# B&R Automation Studio project Y4_V3_1 (part 6)

#### Axis2StateCyclic.ld
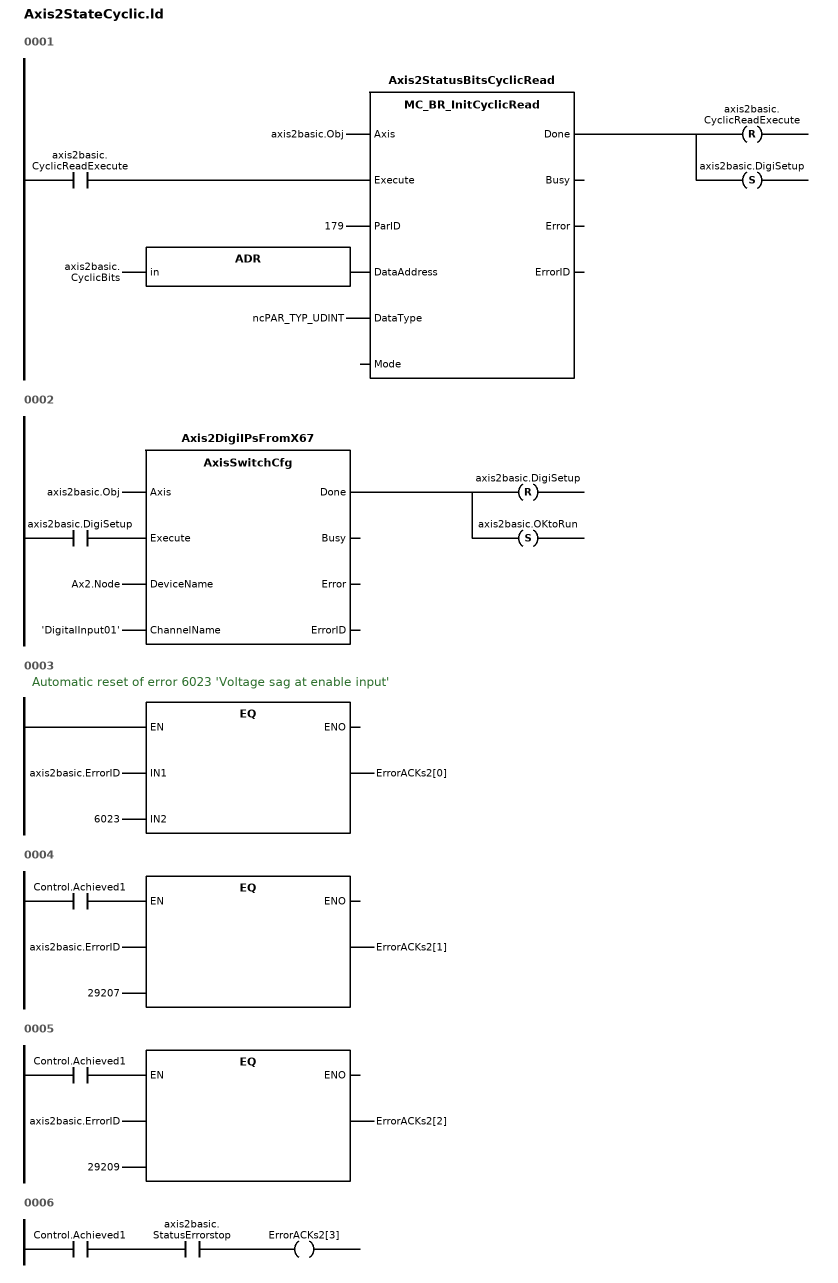
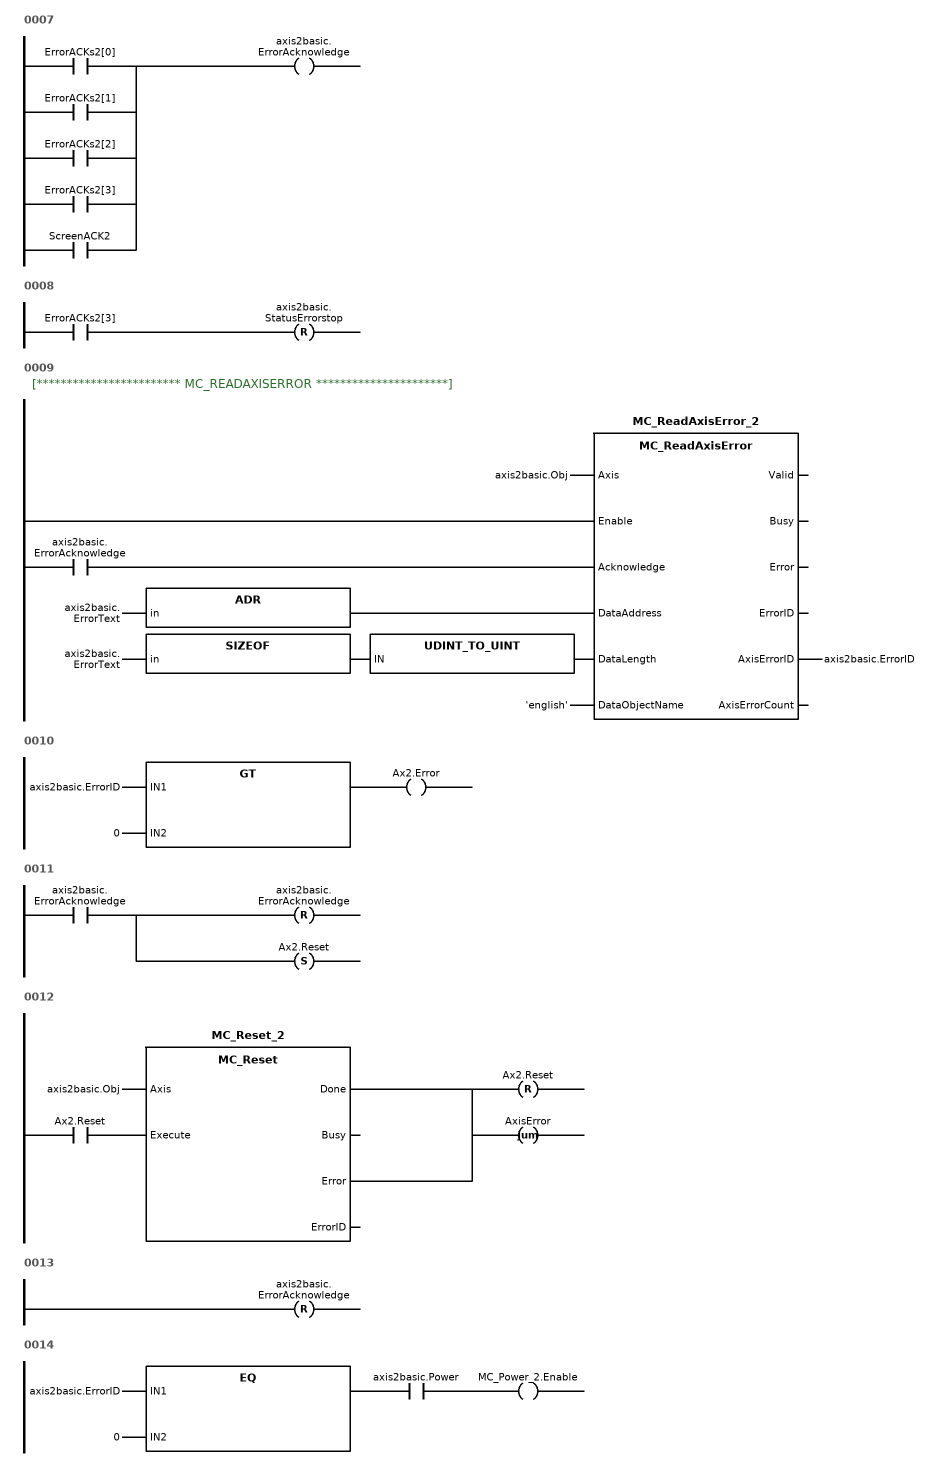
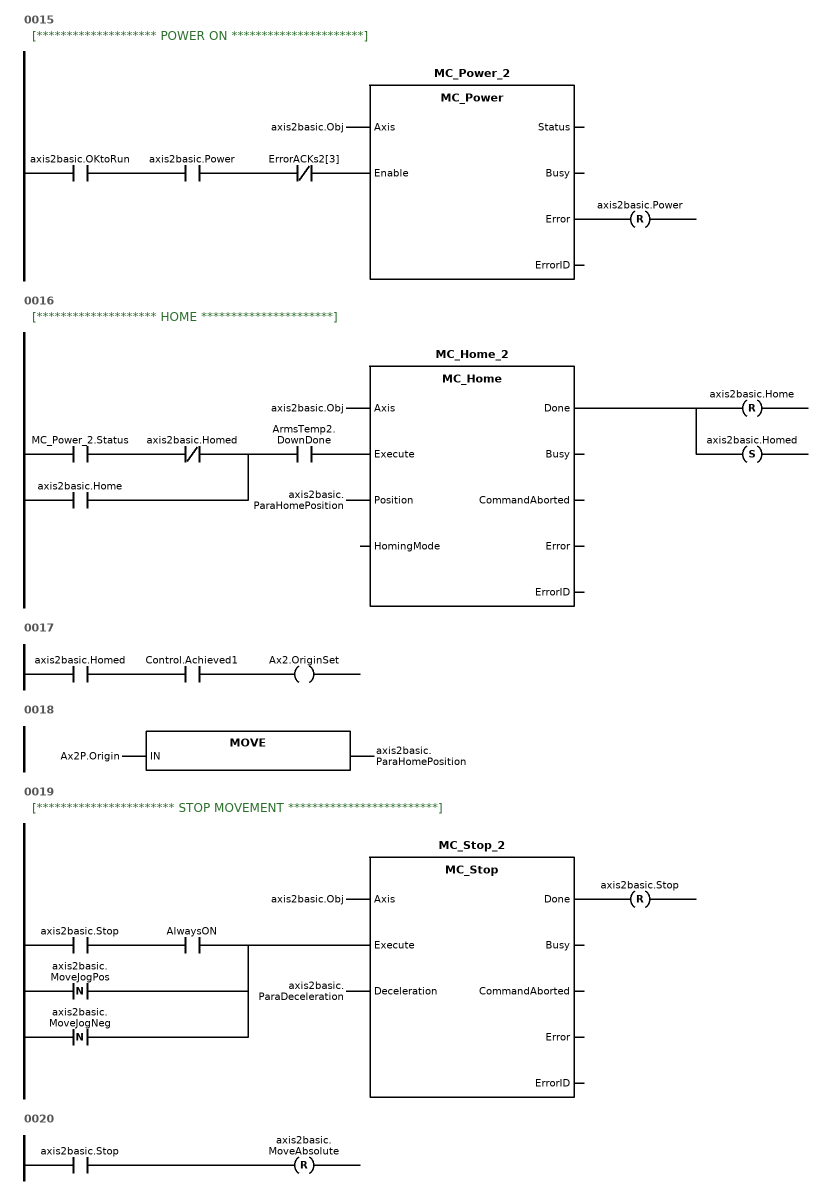
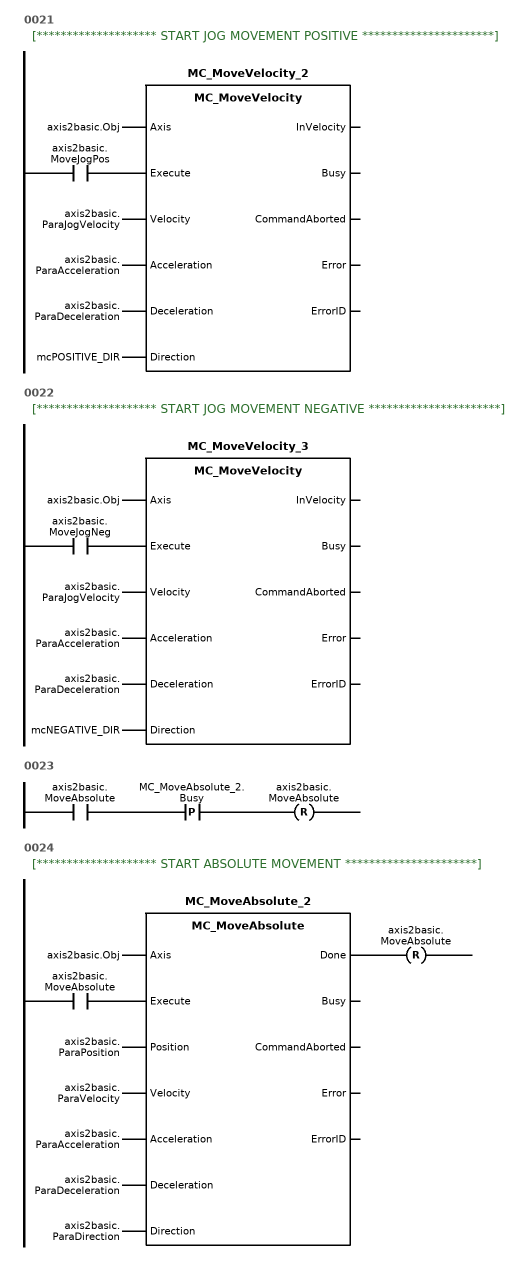
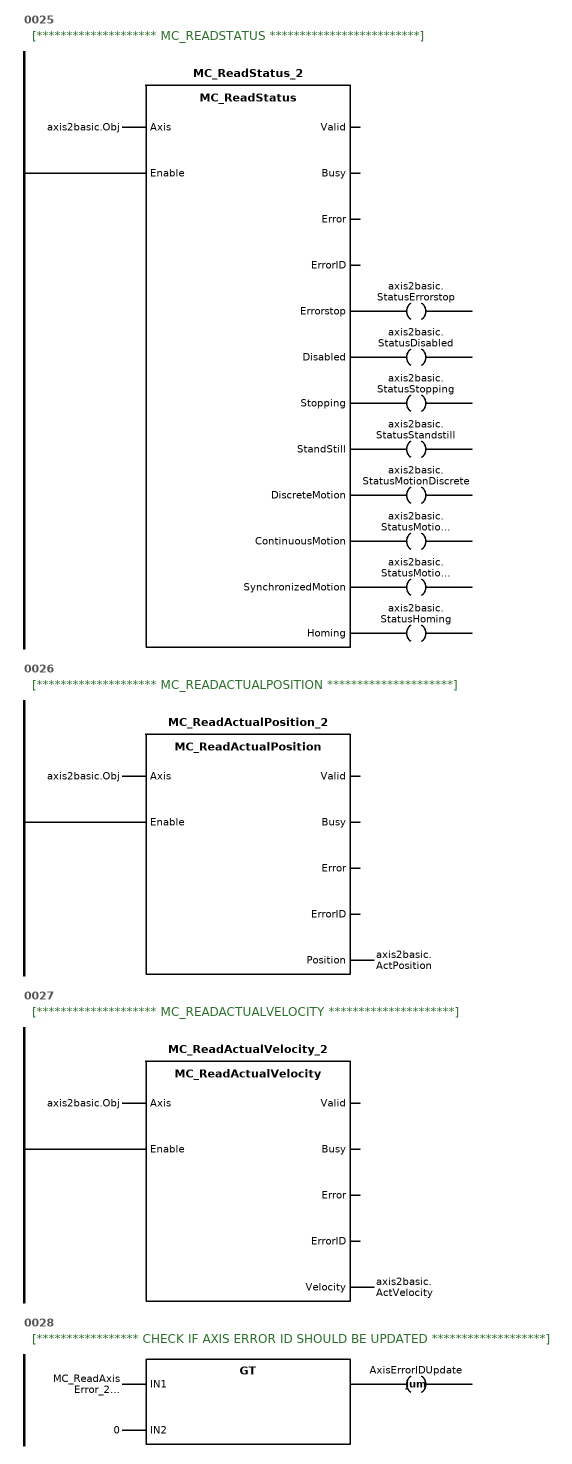
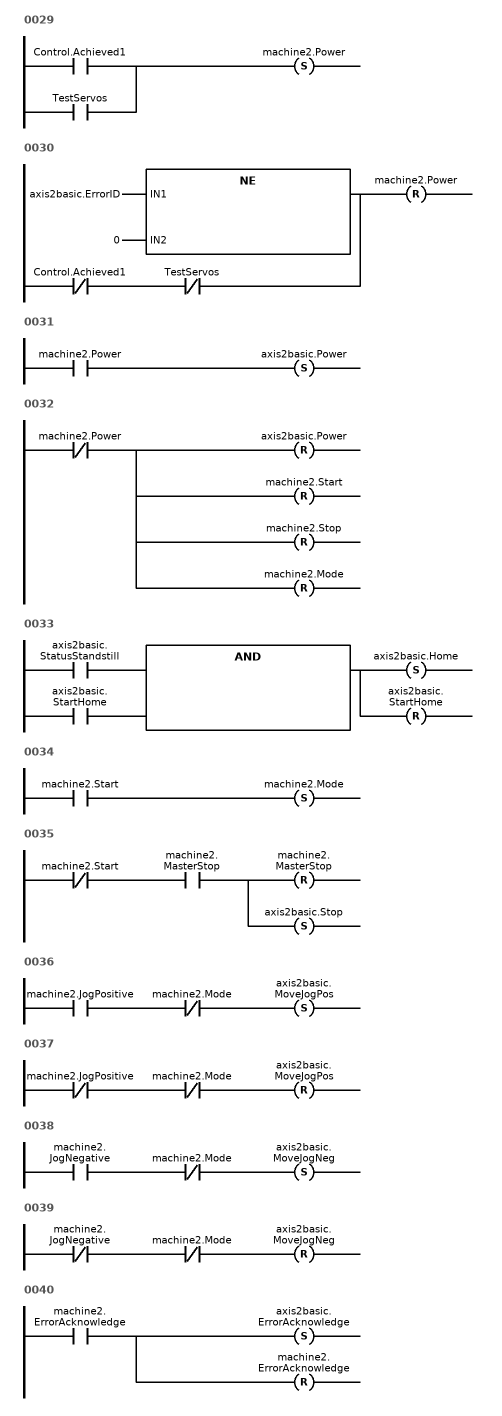
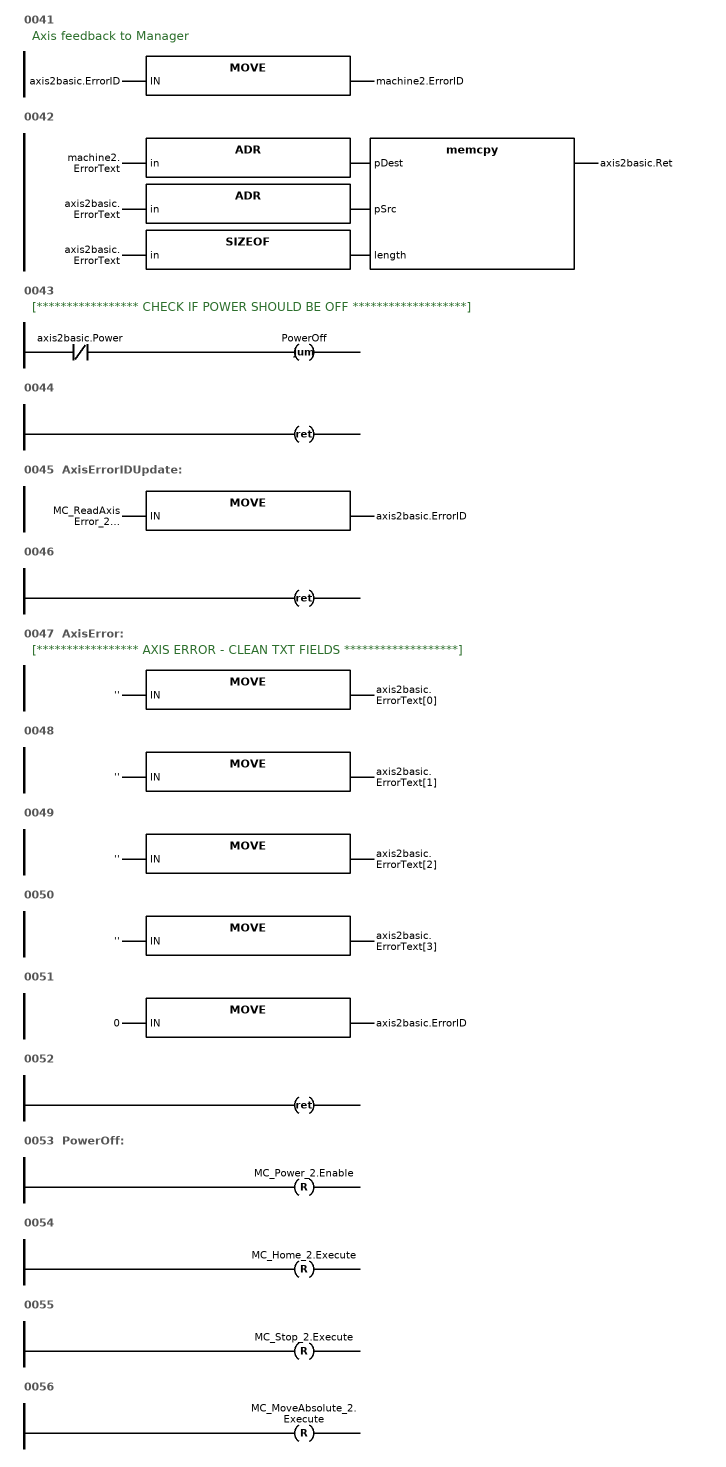
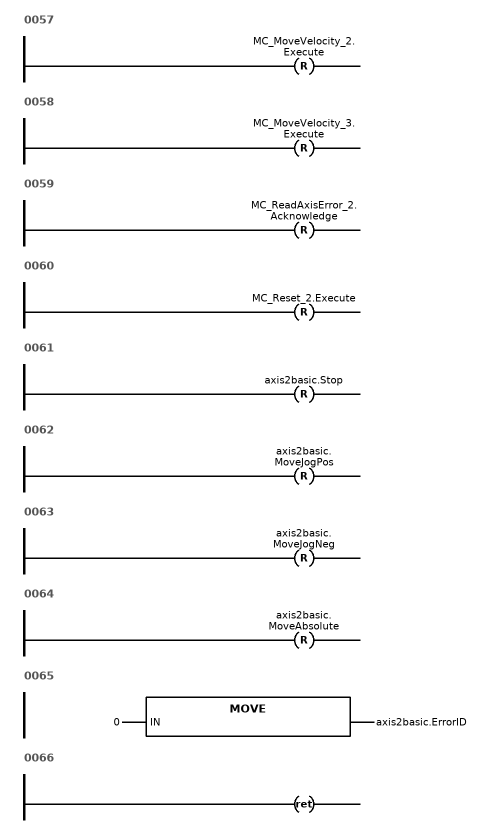
Ladder, written as Structured Text:
```iecst
PROGRAM _CYCLIC
VAR
    _p1 : BOOL;
    _e2 : F_TRIG;
    _e3 : F_TRIG;
    _e4 : R_TRIG;
    _p5 : BOOL;
    _t6 : BOOL;
    _p7 : BOOL;
END_VAR
(* Network 1 *)
Axis2StatusBitsCyclicRead(Axis := axis2basic.Obj, Execute := axis2basic.CyclicReadExecute, ParID := 179, DataAddress := ADR(in := axis2basic.CyclicBits), DataType := ncPAR_TYP_UDINT);
IF Axis2StatusBitsCyclicRead.Done THEN
    axis2basic.CyclicReadExecute := FALSE;
    axis2basic.DigiSetup := TRUE;
END_IF;

(* Network 2 *)
Axis2DigiIPsFromX67(Axis := axis2basic.Obj, Execute := axis2basic.DigiSetup, DeviceName := Ax2.Node, ChannelName := 'DigitalInput01');
IF Axis2DigiIPsFromX67.Done THEN
    axis2basic.DigiSetup := FALSE;
    axis2basic.OKtoRun := TRUE;
END_IF;

(* Network 3: Automatic reset of error 6023 'Voltage sag at enable input' *)
ErrorACKs2[0] := axis2basic.ErrorID = 6023;

(* Network 4 *)
IF Control.Achieved1 THEN ErrorACKs2[1] := axis2basic.ErrorID = 29207; END_IF;

(* Network 5 *)
IF Control.Achieved1 THEN ErrorACKs2[2] := axis2basic.ErrorID = 29209; END_IF;

(* Network 6 *)
ErrorACKs2[3] := Control.Achieved1 AND axis2basic.StatusErrorstop;

(* Network 7 *)
axis2basic.ErrorAcknowledge := ErrorACKs2[0] OR ErrorACKs2[1] OR ErrorACKs2[2] OR ErrorACKs2[3] OR ScreenACK2;

(* Network 8 *)
IF ErrorACKs2[3] THEN axis2basic.StatusErrorstop := FALSE; END_IF;

(* Network 9: [************************ MC_READAXISERROR **********************] *)
MC_ReadAxisError_2(Axis := axis2basic.Obj, Enable := TRUE, Acknowledge := axis2basic.ErrorAcknowledge, DataAddress := ADR(in := axis2basic.ErrorText), DataLength := UDINT_TO_UINT(SIZEOF(in := axis2basic.ErrorText)), DataObjectName := 'english');
axis2basic.ErrorID := MC_ReadAxisError_2.AxisErrorID;

(* Network 10 *)
Ax2.Error := axis2basic.ErrorID > 0;

(* Network 11 *)
_p1 := axis2basic.ErrorAcknowledge;
IF axis2basic.ErrorAcknowledge THEN axis2basic.ErrorAcknowledge := FALSE; END_IF;
IF _p1 THEN Ax2.Reset := TRUE; END_IF;

(* Network 12 *)
MC_Reset_2(Axis := axis2basic.Obj, Execute := Ax2.Reset);
IF MC_Reset_2.Done OR MC_Reset_2.Error THEN
    Ax2.Reset := FALSE;
    JMP AxisError;
END_IF;

(* Network 13 *)
axis2basic.ErrorAcknowledge := FALSE;

(* Network 14 *)
MC_Power_2.Enable := (axis2basic.ErrorID = 0) AND axis2basic.Power;

(* Network 15: [******************** POWER ON **********************] *)
MC_Power_2(Axis := axis2basic.Obj, Enable := axis2basic.OKtoRun AND axis2basic.Power AND NOT ErrorACKs2[3]);
IF MC_Power_2.Error THEN axis2basic.Power := FALSE; END_IF;

(* Network 16: [******************** HOME **********************] *)
MC_Home_2(Axis := axis2basic.Obj, Execute := ((MC_Power_2.Status AND NOT axis2basic.Homed) OR axis2basic.Home) AND ArmsTemp2.DownDone, Position := axis2basic.ParaHomePosition);
IF MC_Home_2.Done THEN
    axis2basic.Home := FALSE;
    axis2basic.Homed := TRUE;
END_IF;

(* Network 17 *)
Ax2.OriginSet := axis2basic.Homed AND Control.Achieved1;

(* Network 18 *)
axis2basic.ParaHomePosition := Ax2P.Origin;

(* Network 19: [*********************** STOP MOVEMENT *************************] *)
_e2(CLK := axis2basic.MoveJogPos);
_e3(CLK := axis2basic.MoveJogNeg);
MC_Stop_2(Axis := axis2basic.Obj, Execute := (axis2basic.Stop AND AlwaysON) OR _e2.Q OR _e3.Q, Deceleration := axis2basic.ParaDeceleration);
IF MC_Stop_2.Done THEN axis2basic.Stop := FALSE; END_IF;

(* Network 20 *)
IF axis2basic.Stop THEN axis2basic.MoveAbsolute := FALSE; END_IF;

(* Network 21: [******************** START JOG MOVEMENT POSITIVE **********************] *)
MC_MoveVelocity_2(Axis := axis2basic.Obj, Execute := axis2basic.MoveJogPos, Velocity := axis2basic.ParaJogVelocity, Acceleration := axis2basic.ParaAcceleration, Deceleration := axis2basic.ParaDeceleration, Direction := mcPOSITIVE_DIR);

(* Network 22: [******************** START JOG MOVEMENT NEGATIVE **********************] *)
MC_MoveVelocity_3(Axis := axis2basic.Obj, Execute := axis2basic.MoveJogNeg, Velocity := axis2basic.ParaJogVelocity, Acceleration := axis2basic.ParaAcceleration, Deceleration := axis2basic.ParaDeceleration, Direction := mcNEGATIVE_DIR);

(* Network 23 *)
_e4(CLK := MC_MoveAbsolute_2.Busy);
IF axis2basic.MoveAbsolute AND _e4.Q THEN axis2basic.MoveAbsolute := FALSE; END_IF;

(* Network 24: [******************** START ABSOLUTE MOVEMENT **********************] *)
MC_MoveAbsolute_2(Axis := axis2basic.Obj, Execute := axis2basic.MoveAbsolute, Position := axis2basic.ParaPosition, Velocity := axis2basic.ParaVelocity, Acceleration := axis2basic.ParaAcceleration, Deceleration := axis2basic.ParaDeceleration, Direction := axis2basic.ParaDirection);
IF MC_MoveAbsolute_2.Done THEN axis2basic.MoveAbsolute := FALSE; END_IF;

(* Network 25: [******************** MC_READSTATUS *************************] *)
MC_ReadStatus_2(Axis := axis2basic.Obj, Enable := TRUE);
axis2basic.StatusErrorstop := MC_ReadStatus_2.Errorstop;
axis2basic.StatusDisabled := MC_ReadStatus_2.Disabled;
axis2basic.StatusStopping := MC_ReadStatus_2.Stopping;
axis2basic.StatusStandstill := MC_ReadStatus_2.StandStill;
axis2basic.StatusMotionDiscrete := MC_ReadStatus_2.DiscreteMotion;
axis2basic.StatusMotionContinous := MC_ReadStatus_2.ContinuousMotion;
axis2basic.StatusMotionSynchronized := MC_ReadStatus_2.SynchronizedMotion;
axis2basic.StatusHoming := MC_ReadStatus_2.Homing;

(* Network 26: [******************** MC_READACTUALPOSITION *********************] *)
MC_ReadActualPosition_2(Axis := axis2basic.Obj, Enable := TRUE);
axis2basic.ActPosition := MC_ReadActualPosition_2.Position;

(* Network 27: [******************** MC_READACTUALVELOCITY *********************] *)
MC_ReadActualVelocity_2(Axis := axis2basic.Obj, Enable := TRUE);
axis2basic.ActVelocity := MC_ReadActualVelocity_2.Velocity;

(* Network 28: [***************** CHECK IF AXIS ERROR ID SHOULD BE UPDATED *******************] *)
IF MC_ReadAxisError_2.AxisErrorID > 0 THEN JMP AxisErrorIDUpdate; END_IF;

(* Network 29 *)
IF Control.Achieved1 OR TestServos THEN machine2.Power := TRUE; END_IF;

(* Network 30 *)
IF (NOT Control.Achieved1 AND NOT TestServos) OR (axis2basic.ErrorID <> 0) THEN
    machine2.Power := FALSE;
END_IF;

(* Network 31 *)
IF machine2.Power THEN axis2basic.Power := TRUE; END_IF;

(* Network 32 *)
IF NOT machine2.Power THEN axis2basic.Power := FALSE; END_IF;
_p5 := NOT machine2.Power;
IF NOT machine2.Power THEN machine2.Start := FALSE; END_IF;
IF _p5 THEN
    machine2.Stop := FALSE;
    machine2.Mode := FALSE;
END_IF;

(* Network 33 *)
_t6 := axis2basic.StatusStandstill AND axis2basic.StartHome;
IF _t6 THEN
    axis2basic.Home := TRUE;
    axis2basic.StartHome := FALSE;
END_IF;

(* Network 34 *)
IF machine2.Start THEN machine2.Mode := TRUE; END_IF;

(* Network 35 *)
_p7 := NOT machine2.Start AND machine2.MasterStop;
IF NOT machine2.Start AND machine2.MasterStop THEN machine2.MasterStop := FALSE; END_IF;
IF _p7 THEN axis2basic.Stop := TRUE; END_IF;

(* Network 36 *)
IF machine2.JogPositive AND NOT machine2.Mode THEN axis2basic.MoveJogPos := TRUE; END_IF;

(* Network 37 *)
IF NOT machine2.JogPositive AND NOT machine2.Mode THEN axis2basic.MoveJogPos := FALSE; END_IF;

(* Network 38 *)
IF machine2.JogNegative AND NOT machine2.Mode THEN axis2basic.MoveJogNeg := TRUE; END_IF;

(* Network 39 *)
IF NOT machine2.JogNegative AND NOT machine2.Mode THEN axis2basic.MoveJogNeg := FALSE; END_IF;

(* Network 40 *)
IF machine2.ErrorAcknowledge THEN
    axis2basic.ErrorAcknowledge := TRUE;
    machine2.ErrorAcknowledge := FALSE;
END_IF;

(* Network 41: Axis feedback to Manager *)
machine2.ErrorID := axis2basic.ErrorID;

(* Network 42 *)
axis2basic.Ret := memcpy(pDest := ADR(in := machine2.ErrorText), pSrc := ADR(in := axis2basic.ErrorText), length := SIZEOF(in := axis2basic.ErrorText));

(* Network 43: [***************** CHECK IF POWER SHOULD BE OFF *******************] *)
IF NOT axis2basic.Power THEN JMP PowerOff; END_IF;

(* Network 44 *)
RETURN;

(* Network 45 *)
AxisErrorIDUpdate:
axis2basic.ErrorID := MC_ReadAxisError_2.AxisErrorID;

(* Network 46 *)
RETURN;

(* Network 47: [***************** AXIS ERROR - CLEAN TXT FIELDS *******************] *)
AxisError:
axis2basic.ErrorText[0] := '';

(* Network 48 *)
axis2basic.ErrorText[1] := '';

(* Network 49 *)
axis2basic.ErrorText[2] := '';

(* Network 50 *)
axis2basic.ErrorText[3] := '';

(* Network 51 *)
axis2basic.ErrorID := 0;

(* Network 52 *)
RETURN;

(* Network 53 *)
PowerOff:
MC_Power_2.Enable := FALSE;

(* Network 54 *)
MC_Home_2.Execute := FALSE;

(* Network 55 *)
MC_Stop_2.Execute := FALSE;

(* Network 56 *)
MC_MoveAbsolute_2.Execute := FALSE;

(* Network 57 *)
MC_MoveVelocity_2.Execute := FALSE;

(* Network 58 *)
MC_MoveVelocity_3.Execute := FALSE;

(* Network 59 *)
MC_ReadAxisError_2.Acknowledge := FALSE;

(* Network 60 *)
MC_Reset_2.Execute := FALSE;

(* Network 61 *)
axis2basic.Stop := FALSE;

(* Network 62 *)
axis2basic.MoveJogPos := FALSE;

(* Network 63 *)
axis2basic.MoveJogNeg := FALSE;

(* Network 64 *)
axis2basic.MoveAbsolute := FALSE;

(* Network 65 *)
axis2basic.ErrorID := 0;

(* Network 66 *)
RETURN;
END_PROGRAM
```

### Program Logical/Motion/Axis3State (IEC)

#### Axis3StateInit.ld
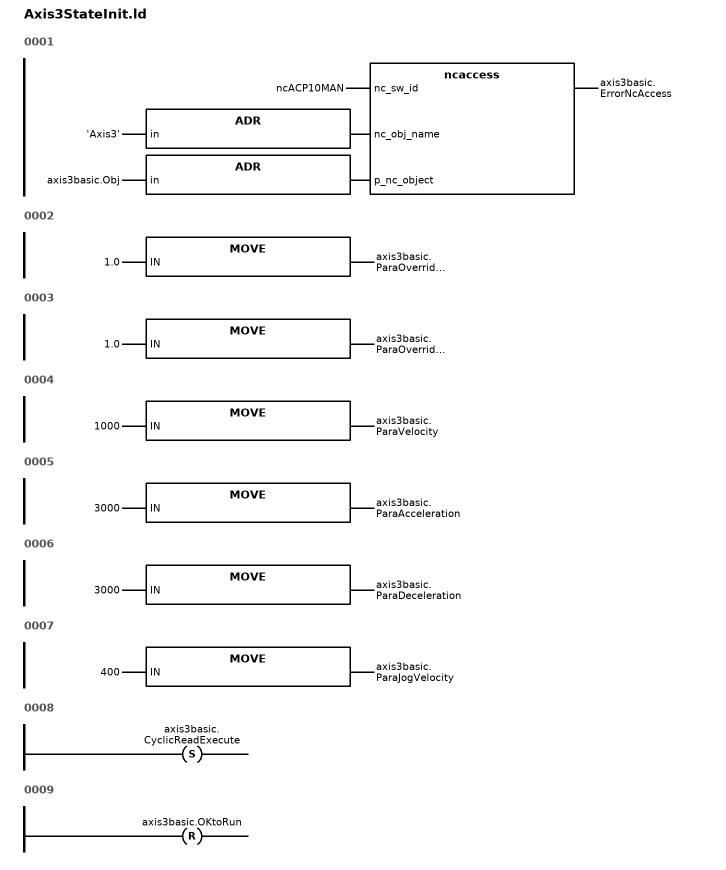
Ladder, written as Structured Text:
```iecst
PROGRAM _INIT
(* Network 1 *)
axis3basic.ErrorNcAccess := ncaccess(nc_sw_id := ncACP10MAN, nc_obj_name := ADR(in := 'Axis3'), p_nc_object := ADR(in := axis3basic.Obj));

(* Network 2 *)
axis3basic.ParaOverrideVelocity := 1.0;

(* Network 3 *)
axis3basic.ParaOverrideAcceleration := 1.0;

(* Network 4 *)
axis3basic.ParaVelocity := 1000;

(* Network 5 *)
axis3basic.ParaAcceleration := 3000;

(* Network 6 *)
axis3basic.ParaDeceleration := 3000;

(* Network 7 *)
axis3basic.ParaJogVelocity := 400;

(* Network 8 *)
axis3basic.CyclicReadExecute := TRUE;

(* Network 9 *)
axis3basic.OKtoRun := FALSE;
END_PROGRAM
```

#### Axis3StateCyclic.ld
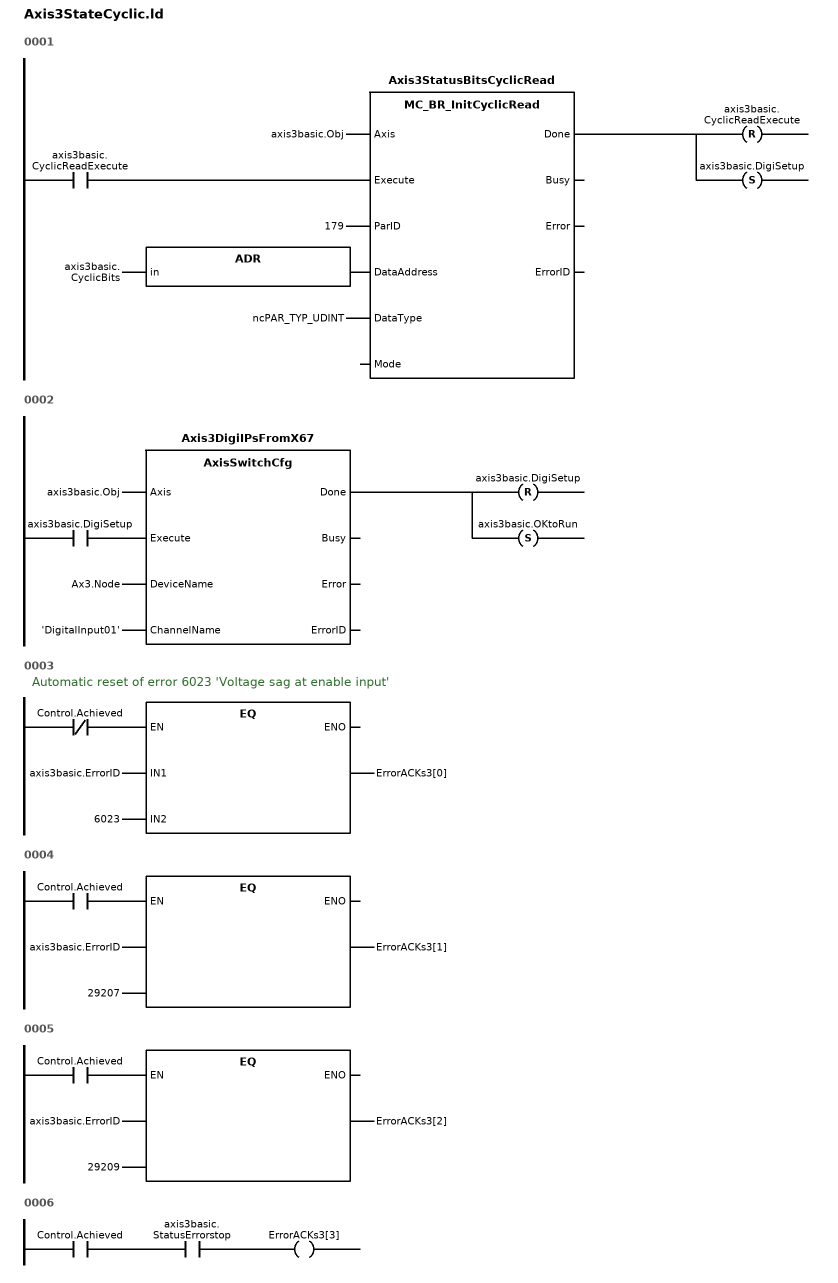
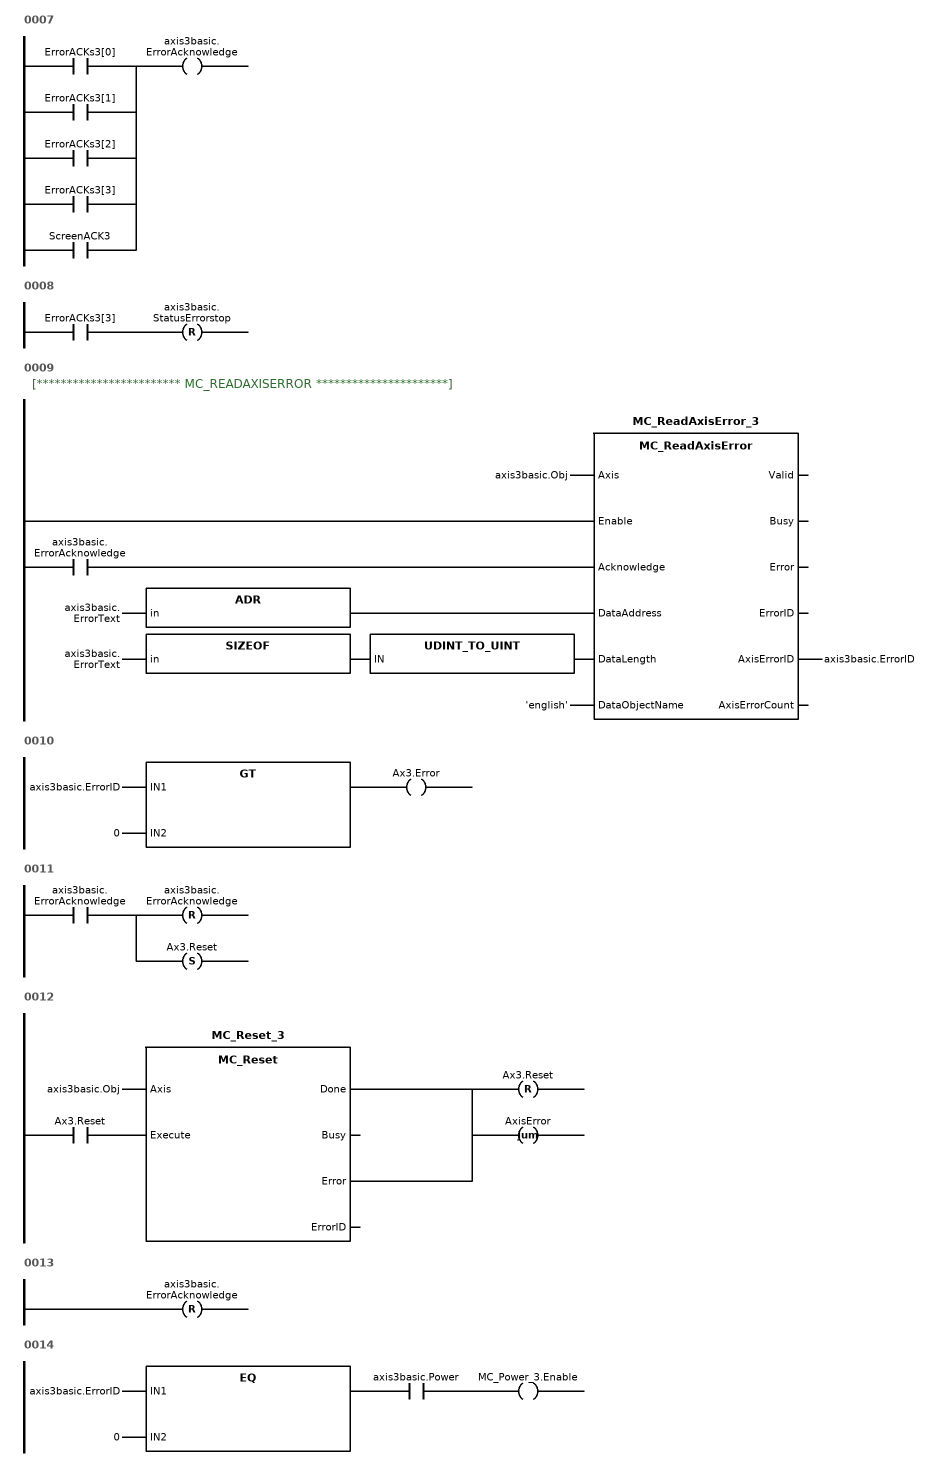
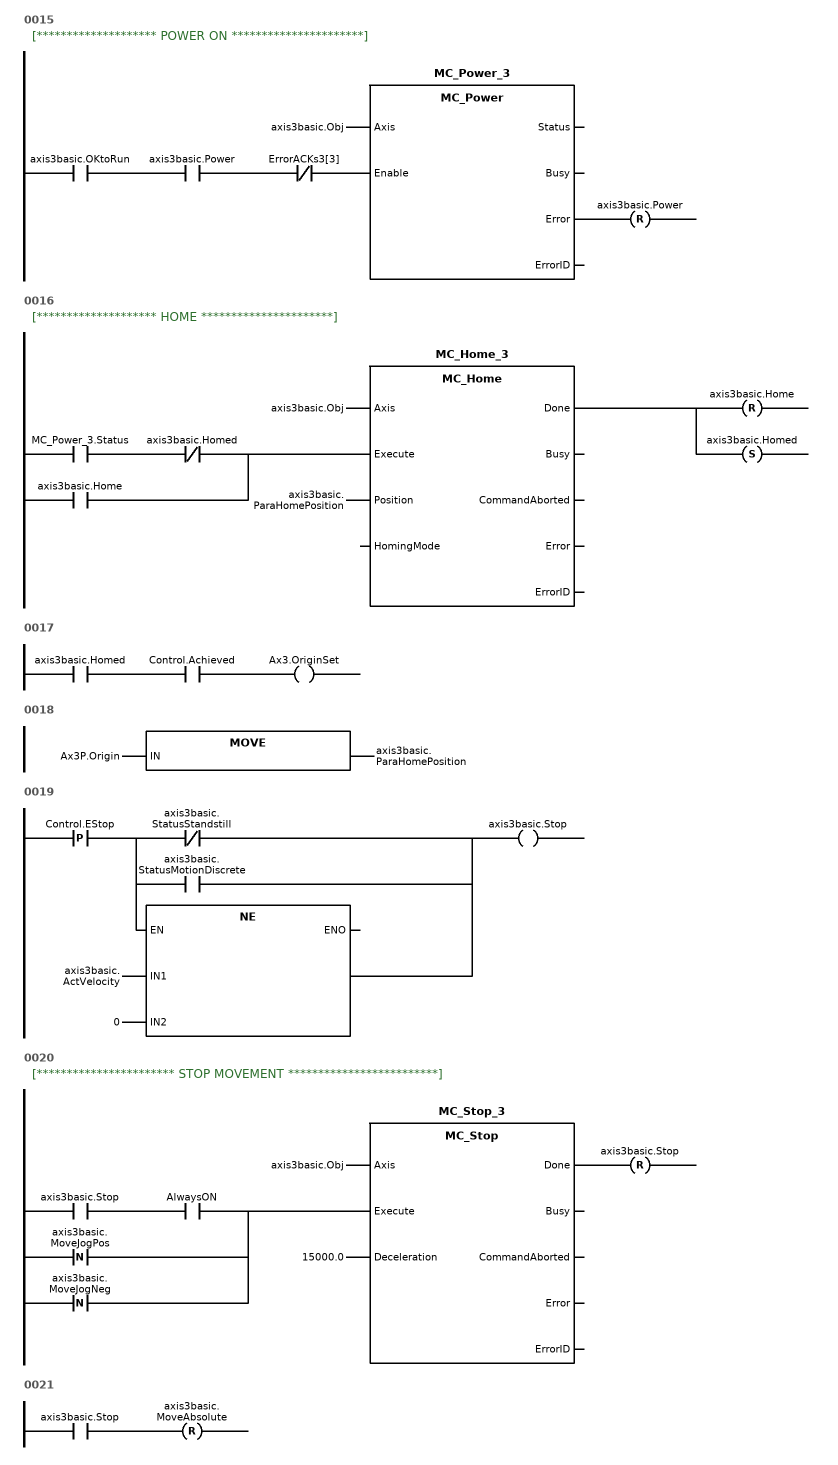
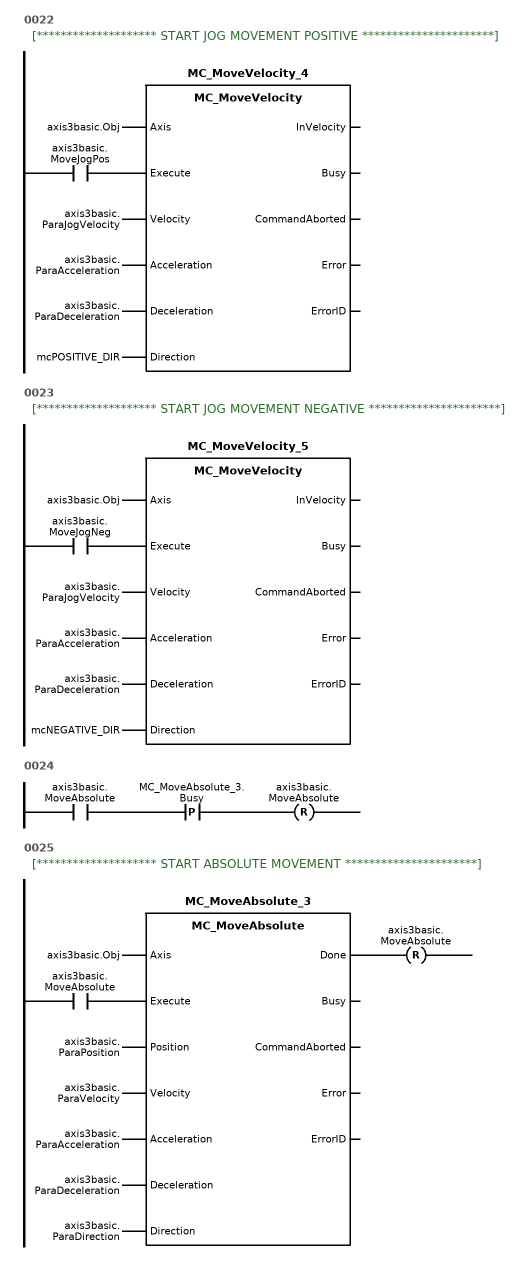
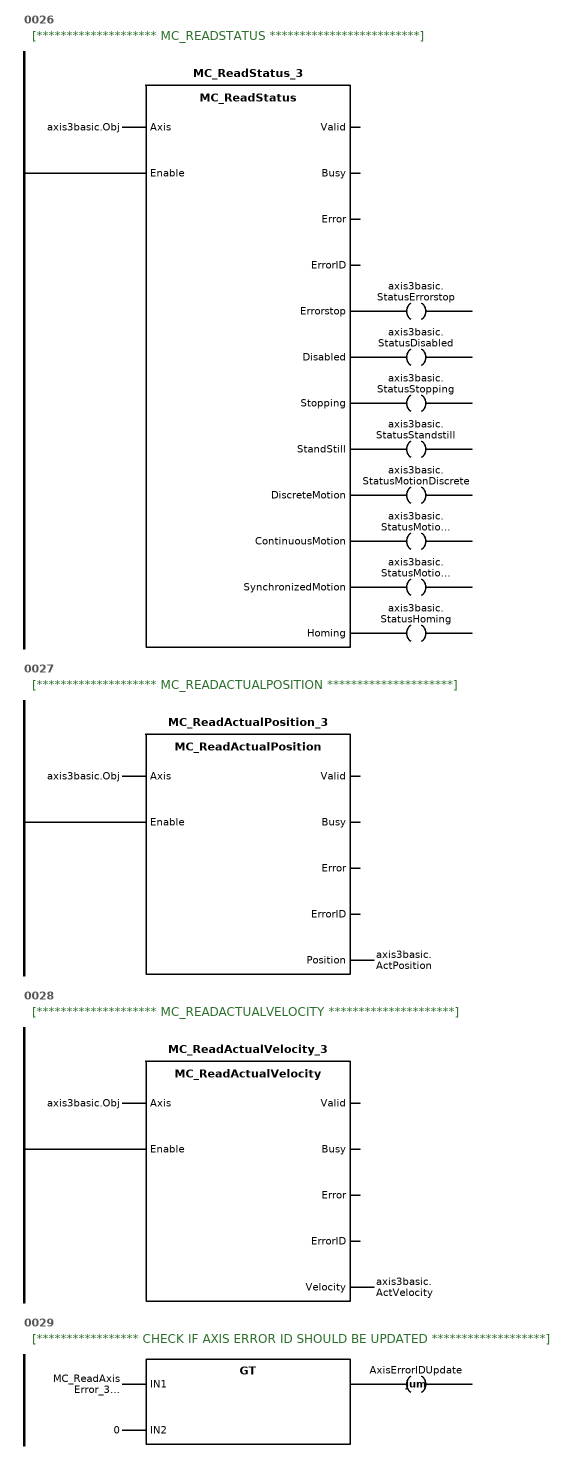
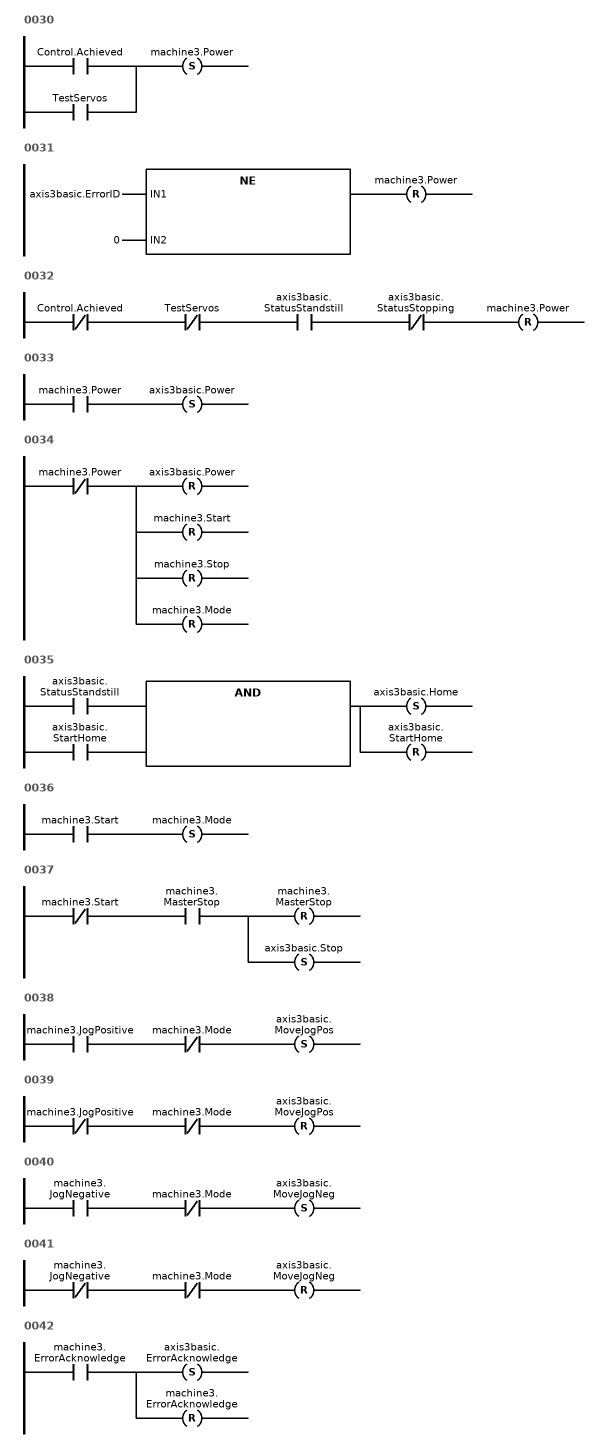
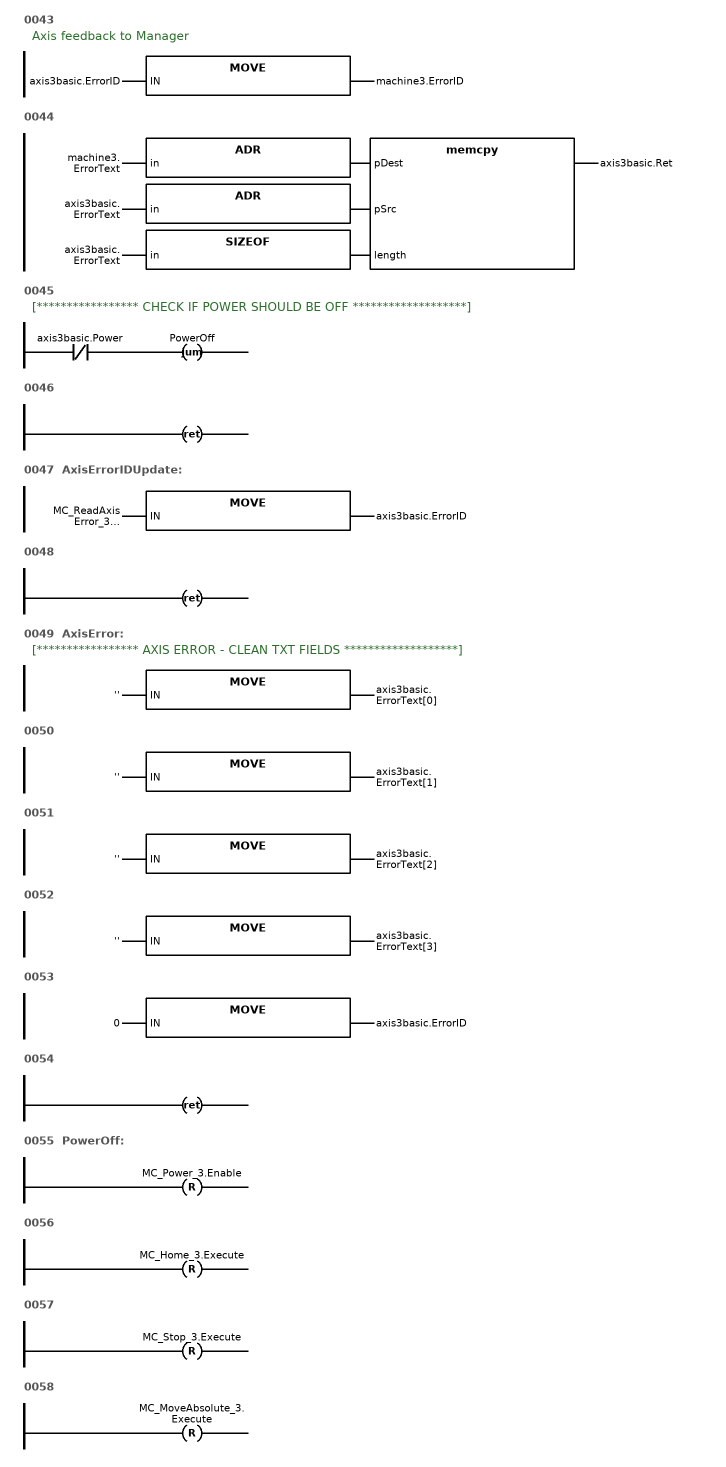
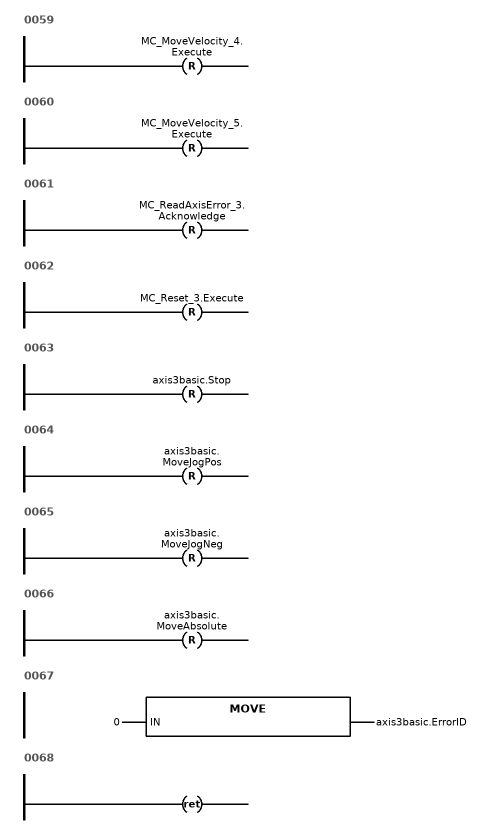
Ladder, written as Structured Text:
```iecst
PROGRAM _CYCLIC
VAR
    _p1 : BOOL;
    _e2 : R_TRIG;
    _t3 : BOOL;
    _e4 : F_TRIG;
    _e5 : F_TRIG;
    _e6 : R_TRIG;
    _p7 : BOOL;
    _t8 : BOOL;
    _p9 : BOOL;
END_VAR
(* Network 1 *)
Axis3StatusBitsCyclicRead(Axis := axis3basic.Obj, Execute := axis3basic.CyclicReadExecute, ParID := 179, DataAddress := ADR(in := axis3basic.CyclicBits), DataType := ncPAR_TYP_UDINT);
IF Axis3StatusBitsCyclicRead.Done THEN
    axis3basic.CyclicReadExecute := FALSE;
    axis3basic.DigiSetup := TRUE;
END_IF;

(* Network 2 *)
Axis3DigiIPsFromX67(Axis := axis3basic.Obj, Execute := axis3basic.DigiSetup, DeviceName := Ax3.Node, ChannelName := 'DigitalInput01');
IF Axis3DigiIPsFromX67.Done THEN
    axis3basic.DigiSetup := FALSE;
    axis3basic.OKtoRun := TRUE;
END_IF;

(* Network 3: Automatic reset of error 6023 'Voltage sag at enable input' *)
IF NOT Control.Achieved THEN ErrorACKs3[0] := axis3basic.ErrorID = 6023; END_IF;

(* Network 4 *)
IF Control.Achieved THEN ErrorACKs3[1] := axis3basic.ErrorID = 29207; END_IF;

(* Network 5 *)
IF Control.Achieved THEN ErrorACKs3[2] := axis3basic.ErrorID = 29209; END_IF;

(* Network 6 *)
ErrorACKs3[3] := Control.Achieved AND axis3basic.StatusErrorstop;

(* Network 7 *)
axis3basic.ErrorAcknowledge := ErrorACKs3[0] OR ErrorACKs3[1] OR ErrorACKs3[2] OR ErrorACKs3[3] OR ScreenACK3;

(* Network 8 *)
IF ErrorACKs3[3] THEN axis3basic.StatusErrorstop := FALSE; END_IF;

(* Network 9: [************************ MC_READAXISERROR **********************] *)
MC_ReadAxisError_3(Axis := axis3basic.Obj, Enable := TRUE, Acknowledge := axis3basic.ErrorAcknowledge, DataAddress := ADR(in := axis3basic.ErrorText), DataLength := UDINT_TO_UINT(SIZEOF(in := axis3basic.ErrorText)), DataObjectName := 'english');
axis3basic.ErrorID := MC_ReadAxisError_3.AxisErrorID;

(* Network 10 *)
Ax3.Error := axis3basic.ErrorID > 0;

(* Network 11 *)
_p1 := axis3basic.ErrorAcknowledge;
IF axis3basic.ErrorAcknowledge THEN axis3basic.ErrorAcknowledge := FALSE; END_IF;
IF _p1 THEN Ax3.Reset := TRUE; END_IF;

(* Network 12 *)
MC_Reset_3(Axis := axis3basic.Obj, Execute := Ax3.Reset);
IF MC_Reset_3.Done OR MC_Reset_3.Error THEN
    Ax3.Reset := FALSE;
    JMP AxisError;
END_IF;

(* Network 13 *)
axis3basic.ErrorAcknowledge := FALSE;

(* Network 14 *)
MC_Power_3.Enable := (axis3basic.ErrorID = 0) AND axis3basic.Power;

(* Network 15: [******************** POWER ON **********************] *)
MC_Power_3(Axis := axis3basic.Obj, Enable := axis3basic.OKtoRun AND axis3basic.Power AND NOT ErrorACKs3[3]);
IF MC_Power_3.Error THEN axis3basic.Power := FALSE; END_IF;

(* Network 16: [******************** HOME **********************] *)
MC_Home_3(Axis := axis3basic.Obj, Execute := (MC_Power_3.Status AND NOT axis3basic.Homed) OR axis3basic.Home, Position := axis3basic.ParaHomePosition);
IF MC_Home_3.Done THEN
    axis3basic.Home := FALSE;
    axis3basic.Homed := TRUE;
END_IF;

(* Network 17 *)
Ax3.OriginSet := axis3basic.Homed AND Control.Achieved;

(* Network 18 *)
axis3basic.ParaHomePosition := Ax3P.Origin;

(* Network 19 *)
_e2(CLK := Control.EStop);
IF _e2.Q THEN _t3 := axis3basic.ActVelocity <> 0; END_IF;
axis3basic.Stop := (_e2.Q AND (NOT axis3basic.StatusStandstill OR axis3basic.StatusMotionDiscrete)) OR _t3;

(* Network 20: [*********************** STOP MOVEMENT *************************] *)
_e4(CLK := axis3basic.MoveJogPos);
_e5(CLK := axis3basic.MoveJogNeg);
MC_Stop_3(Axis := axis3basic.Obj, Execute := (axis3basic.Stop AND AlwaysON) OR _e4.Q OR _e5.Q, Deceleration := 15000.0);
IF MC_Stop_3.Done THEN axis3basic.Stop := FALSE; END_IF;

(* Network 21 *)
IF axis3basic.Stop THEN axis3basic.MoveAbsolute := FALSE; END_IF;

(* Network 22: [******************** START JOG MOVEMENT POSITIVE **********************] *)
MC_MoveVelocity_4(Axis := axis3basic.Obj, Execute := axis3basic.MoveJogPos, Velocity := axis3basic.ParaJogVelocity, Acceleration := axis3basic.ParaAcceleration, Deceleration := axis3basic.ParaDeceleration, Direction := mcPOSITIVE_DIR);

(* Network 23: [******************** START JOG MOVEMENT NEGATIVE **********************] *)
MC_MoveVelocity_5(Axis := axis3basic.Obj, Execute := axis3basic.MoveJogNeg, Velocity := axis3basic.ParaJogVelocity, Acceleration := axis3basic.ParaAcceleration, Deceleration := axis3basic.ParaDeceleration, Direction := mcNEGATIVE_DIR);

(* Network 24 *)
_e6(CLK := MC_MoveAbsolute_3.Busy);
IF axis3basic.MoveAbsolute AND _e6.Q THEN axis3basic.MoveAbsolute := FALSE; END_IF;

(* Network 25: [******************** START ABSOLUTE MOVEMENT **********************] *)
MC_MoveAbsolute_3(Axis := axis3basic.Obj, Execute := axis3basic.MoveAbsolute, Position := axis3basic.ParaPosition, Velocity := axis3basic.ParaVelocity, Acceleration := axis3basic.ParaAcceleration, Deceleration := axis3basic.ParaDeceleration, Direction := axis3basic.ParaDirection);
IF MC_MoveAbsolute_3.Done THEN axis3basic.MoveAbsolute := FALSE; END_IF;

(* Network 26: [******************** MC_READSTATUS *************************] *)
MC_ReadStatus_3(Axis := axis3basic.Obj, Enable := TRUE);
axis3basic.StatusErrorstop := MC_ReadStatus_3.Errorstop;
axis3basic.StatusDisabled := MC_ReadStatus_3.Disabled;
axis3basic.StatusStopping := MC_ReadStatus_3.Stopping;
axis3basic.StatusStandstill := MC_ReadStatus_3.StandStill;
axis3basic.StatusMotionDiscrete := MC_ReadStatus_3.DiscreteMotion;
axis3basic.StatusMotionContinous := MC_ReadStatus_3.ContinuousMotion;
axis3basic.StatusMotionSynchronized := MC_ReadStatus_3.SynchronizedMotion;
axis3basic.StatusHoming := MC_ReadStatus_3.Homing;

(* Network 27: [******************** MC_READACTUALPOSITION *********************] *)
MC_ReadActualPosition_3(Axis := axis3basic.Obj, Enable := TRUE);
axis3basic.ActPosition := MC_ReadActualPosition_3.Position;

(* Network 28: [******************** MC_READACTUALVELOCITY *********************] *)
MC_ReadActualVelocity_3(Axis := axis3basic.Obj, Enable := TRUE);
axis3basic.ActVelocity := MC_ReadActualVelocity_3.Velocity;

(* Network 29: [***************** CHECK IF AXIS ERROR ID SHOULD BE UPDATED *******************] *)
IF MC_ReadAxisError_3.AxisErrorID > 0 THEN JMP AxisErrorIDUpdate; END_IF;

(* Network 30 *)
IF Control.Achieved OR TestServos THEN machine3.Power := TRUE; END_IF;

(* Network 31 *)
IF axis3basic.ErrorID <> 0 THEN machine3.Power := FALSE; END_IF;

(* Network 32 *)
IF NOT Control.Achieved AND NOT TestServos AND axis3basic.StatusStandstill AND NOT axis3basic.StatusStopping THEN
    machine3.Power := FALSE;
END_IF;

(* Network 33 *)
IF machine3.Power THEN axis3basic.Power := TRUE; END_IF;

(* Network 34 *)
IF NOT machine3.Power THEN axis3basic.Power := FALSE; END_IF;
_p7 := NOT machine3.Power;
IF NOT machine3.Power THEN machine3.Start := FALSE; END_IF;
IF _p7 THEN
    machine3.Stop := FALSE;
    machine3.Mode := FALSE;
END_IF;

(* Network 35 *)
_t8 := axis3basic.StatusStandstill AND axis3basic.StartHome;
IF _t8 THEN
    axis3basic.Home := TRUE;
    axis3basic.StartHome := FALSE;
END_IF;

(* Network 36 *)
IF machine3.Start THEN machine3.Mode := TRUE; END_IF;

(* Network 37 *)
_p9 := NOT machine3.Start AND machine3.MasterStop;
IF NOT machine3.Start AND machine3.MasterStop THEN machine3.MasterStop := FALSE; END_IF;
IF _p9 THEN axis3basic.Stop := TRUE; END_IF;

(* Network 38 *)
IF machine3.JogPositive AND NOT machine3.Mode THEN axis3basic.MoveJogPos := TRUE; END_IF;

(* Network 39 *)
IF NOT machine3.JogPositive AND NOT machine3.Mode THEN axis3basic.MoveJogPos := FALSE; END_IF;

(* Network 40 *)
IF machine3.JogNegative AND NOT machine3.Mode THEN axis3basic.MoveJogNeg := TRUE; END_IF;

(* Network 41 *)
IF NOT machine3.JogNegative AND NOT machine3.Mode THEN axis3basic.MoveJogNeg := FALSE; END_IF;

(* Network 42 *)
IF machine3.ErrorAcknowledge THEN
    axis3basic.ErrorAcknowledge := TRUE;
    machine3.ErrorAcknowledge := FALSE;
END_IF;

(* Network 43: Axis feedback to Manager *)
machine3.ErrorID := axis3basic.ErrorID;

(* Network 44 *)
axis3basic.Ret := memcpy(pDest := ADR(in := machine3.ErrorText), pSrc := ADR(in := axis3basic.ErrorText), length := SIZEOF(in := axis3basic.ErrorText));

(* Network 45: [***************** CHECK IF POWER SHOULD BE OFF *******************] *)
IF NOT axis3basic.Power THEN JMP PowerOff; END_IF;

(* Network 46 *)
RETURN;

(* Network 47 *)
AxisErrorIDUpdate:
axis3basic.ErrorID := MC_ReadAxisError_3.AxisErrorID;

(* Network 48 *)
RETURN;

(* Network 49: [***************** AXIS ERROR - CLEAN TXT FIELDS *******************] *)
AxisError:
axis3basic.ErrorText[0] := '';

(* Network 50 *)
axis3basic.ErrorText[1] := '';

(* Network 51 *)
axis3basic.ErrorText[2] := '';

(* Network 52 *)
axis3basic.ErrorText[3] := '';

(* Network 53 *)
axis3basic.ErrorID := 0;

(* Network 54 *)
RETURN;

(* Network 55 *)
PowerOff:
MC_Power_3.Enable := FALSE;

(* Network 56 *)
MC_Home_3.Execute := FALSE;

(* Network 57 *)
MC_Stop_3.Execute := FALSE;

(* Network 58 *)
MC_MoveAbsolute_3.Execute := FALSE;

(* Network 59 *)
MC_MoveVelocity_4.Execute := FALSE;

(* Network 60 *)
MC_MoveVelocity_5.Execute := FALSE;

(* Network 61 *)
MC_ReadAxisError_3.Acknowledge := FALSE;

(* Network 62 *)
MC_Reset_3.Execute := FALSE;

(* Network 63 *)
axis3basic.Stop := FALSE;

(* Network 64 *)
axis3basic.MoveJogPos := FALSE;

(* Network 65 *)
axis3basic.MoveJogNeg := FALSE;

(* Network 66 *)
axis3basic.MoveAbsolute := FALSE;

(* Network 67 *)
axis3basic.ErrorID := 0;

(* Network 68 *)
RETURN;
END_PROGRAM
```

### Data object Logical/Motion/axis3 (Ax) - ACP10: Axis data object.

#### axis3.ax
```
InitParameter (Version=2.37.0, NcSwId=ACP10)
  ACP10AXIS_typ:
    dig_in:
      level:
        reference = ncACTIV_HI
        pos_hw_end = ncACTIV_LO
        neg_hw_end = ncACTIV_LO
        trigger1 = ncACTIV_HI
        trigger2 = ncACTIV_HI
    encoder_if:
      parameter:
        count_dir = ncSTANDARD
        scaling:
          load:
            units = 1521
            rev_motor = 10
    limit:
      parameter:
        v_pos = 10000
        v_neg = 10000
        a1_pos = 9000.0
        a2_pos = 7000.0
        a1_neg = 9000.0
        a2_neg = 7000.0
        t_jolt = 0
        t_in_pos = 0
        pos_sw_end = 2000000000
        neg_sw_end = -2000000000
        ds_warning = 500
        ds_stop = 1000
        a_stop = 1.0e30
        dv_stop = 0
        dv_stop_mode = ncOFF
    controller:
      mode = ncPOSITION
      position:
        kv = 50
        tn = 0
        t_predict = 0.0008
        t_total = 0.0008
        p_max = 10000
        i_max = 0
      speed:
        kv = 2.0
        tn = 0
        t_filter = 0.0
        isq_filter1:
          type = ncOFF
          a0 = 0.0
          a1 = 0.0
          b0 = 0.0
          b1 = 0.0
          b2 = 0.0
          c0_par_id = 0
          c1_par_id = 0
        isq_filter2:
          type = ncOFF
          a0 = 0.0
          a1 = 0.0
          b0 = 0.0
          b1 = 0.0
          b2 = 0.0
          c0_par_id = 0
          c1_par_id = 0
        isq_filter3:
          type = ncOFF
          a0 = 0.0
          a1 = 0.0
          b0 = 0.0
          b1 = 0.0
          b2 = 0.0
          c0_par_id = 0
          c1_par_id = 0
      uf:
        type = ncLINEAR
        auto_config = ncMOTOR_PAR
        u0 = 0
        un = 0
        fn = 50.0
        k_f_slip = 0
      ff:
        torque_load = 0.0
        torque_pos = 0.0
        torque_neg = 0.0
        kv_torque = 0.0
        inertia = 0.0
        t_filter_a = 0.0
    move:
      stop:
        parameter[0]:
          decel_ramp = ncA_LIMIT
          controller = ncON
        parameter[1]:
          decel_ramp = ncA_LIMIT
          controller = ncON
        parameter[2]:
          decel_ramp = ncA_LIMIT
          controller = ncON
        parameter[3]:
          decel_ramp = ncA_LIMIT
          controller = ncON
        quickstop:
          decel_ramp = ncA_LIMIT
        drive_error:
          decel_ramp = ncA_LIMIT
      homing:
        parameter:
          s = 0
          v_switch = 500.0
          v_trigger = 25.0
          a = 1000.0
          mode = ncSWITCH_GATE
          edge_sw = ncNEGATIVE
          start_dir = ncNEGATIVE
          trigg_dir = ncNEGATIVE
          ref_pulse = ncOFF
          fix_dir = ncOFF
          tr_s_block = 0
          torque_lim = 0
          ds_block = 0
          ds_stop = 0
      basis:
        parameter:
          v_pos = 10000
          v_neg = 10000
          a1_pos = 50000
          a2_pos = 40000.0
          a1_neg = 50000
          a2_neg = 40000.0
    message:
      text:
        parameter:
          format = ncBREAK
          columns = 80
          data_modul = english
```

### Data object Logical/Motion/table_par3 (Apt) - ACOPOS Parameter Table

#### table_par3.apt
```
AcoposParameterTable:
  Root Parameters:
    8JSA54.R0050D000-0 Rev.C0 (StructureEdit=FALSE)  // 8JSA54.R0050D000-0 Rev.C0
      General parameters:
        30 = 0x0002 (Name=MOTOR_TYPE)  // Motor: Type
        31 = 0x0203 (Name=MOTOR_COMPATIBILITY)  // Motor: Software compatibility
        46 = 1 (Name=MOTOR_WIND_CONNECT)  // Motor: Winding connection
        47 = 5 (Name=MOTOR_POLEPAIRS)  // Motor: Number of pole-pairs
      Brake parameters:
        42 = 0 (Name=MOTOR_BRAKE_CURR_RATED, Unit=A)  // Motor holding brake: Rated current
        43 = 0 (Name=MOTOR_BRAKE_TORQ_RATED, Unit=Nm)  // Motor holding brake: Rated torque
        44 = 0 (Name=MOTOR_BRAKE_ON_TIME, Unit=s)  // Motor holding brake: Engaging delay
        45 = 0 (Name=MOTOR_BRAKE_OFF_TIME, Unit=s)  // Motor holding brake: Release delay
      Thermo sensor parameters:
        64 = 632 (Name=MOTOR_TEMPSENS_PAR1)  // Temperature sensor: Parameter 1
        65 = 2225 (Name=MOTOR_TEMPSENS_PAR2)  // Temperature sensor: Parameter 2
        66 = -30 (Name=MOTOR_TEMPSENS_PAR3)  // Temperature sensor: Parameter 3
        67 = 5.7266 (Name=MOTOR_TEMPSENS_PAR4)  // Temperature sensor: Parameter 4
        68 = 36.0938 (Name=MOTOR_TEMPSENS_PAR5)  // Temperature sensor: Parameter 5
        69 = 62.9375 (Name=MOTOR_TEMPSENS_PAR6)  // Temperature sensor: Parameter 6
        70 = 87.25 (Name=MOTOR_TEMPSENS_PAR7)  // Temperature sensor: Parameter 7
        71 = 109.6016 (Name=MOTOR_TEMPSENS_PAR8)  // Temperature sensor: Parameter 8
        72 = 130.3984 (Name=MOTOR_TEMPSENS_PAR9)  // Temperature sensor: Parameter 9
        73 = 150 (Name=MOTOR_TEMPSENS_PAR10)  // Temperature sensor: Parameter 10
        75 = 0 (Name=MOTOR_THERMAL_CONST, Unit=s)  // Motor: Thermal time constant (for MOTOR_COMPATIBILITY 0x0202)
      Motor parameters:
        48 = 560 (Name=MOTOR_VOLTAGE_RATED, Unit=V)  // Motor: Rated voltage
        49 = 73.3 (Name=MOTOR_VOLTAGE_CONST, Unit=mV*min)  // Motor: Voltage constant
        50 = 5000 (Name=MOTOR_SPEED_RATED, Unit=1/min)  // Motor: Rated speed
        51 = 6000 (Name=MOTOR_SPEED_MAX, Unit=1/min)  // Motor: Maximum speed
        52 = 14.1 (Name=MOTOR_TORQ_STALL, Unit=Nm)  // Motor: Stall torque
        53 = 6.92 (Name=MOTOR_TORQ_RATED, Unit=Nm)  // Motor: Rated torque
        54 = 53.7 (Name=MOTOR_TORQ_MAX, Unit=Nm)  // Motor: Peak torque
        55 = 1.13 (Name=MOTOR_TORQ_CONST, Unit=Nm/A)  // Motor: Torque constant
        56 = 12.5 (Name=MOTOR_CURR_STALL, Unit=A)  // Motor: Stall current
        57 = 6.11 (Name=MOTOR_CURR_RATED, Unit=A)  // Motor: Rated current
        58 = 62.5 (Name=MOTOR_CURR_MAX, Unit=A)  // Motor: Peak current
        59 = 1.2973 (Name=MOTOR_WIND_CROSS_SECT, Unit=mm²)  // Motor: Line cross section
        60 = 0.65 (Name=MOTOR_STATOR_RESISTANCE, Unit=Ohm)  // Motor: Stator resistance
        61 = 0.0035 (Name=MOTOR_STATOR_INDUCTANCE, Unit=Henry)  // Motor: Stator inductance
        62 = 0.0012 (Name=MOTOR_INERTIA, Unit=kgm²)  // Motor: Moment of inertia
        63 = 0 (Name=MOTOR_COMMUT_OFFSET, Unit=rad)  // Motor: Commutation offset
        849 = 1860 (Name=MOTOR_TAU_THERM, Unit=s)  // Motor: Thermal time constant
      Isolation parameters:
        74 = 130 (Name=MOTOR_WIND_TEMP_MAX, Unit=°C)  // Temperature sensor: Limit temperature
    SS2 (StructureEdit=FALSE)  // 8AC122.60-3
      97 = ncRESOLVER (Name=ENCOD_TYPE)  // Encoder1: Type
      109 = 4096 (Name=SCALE_ENCOD_INCR)  // Encoder1: Encoder scaling: increments per SCALE_ENCOD_MOTOR_REV motor revolutions
      203 = 1 (Name=ENCOD_POLEPAIRS)  // Encoder1: Resolver polepairs per encoder revolution
      727 = 0 (Name=ENCOD_LINE_CHK_IGNORE)  // Encoder1: Ignore check
      1048 = 0.5 (Name=ENCOD_TRANS_RATIO)  // Encoder1: Resolver transmission ratio
```

### IPConfig.var - Local variables
```iecst
(********************************************************************
 * COPYRIGHT --
 ********************************************************************
 * Program: IPConfig
 * File: IPConfig.var
 * Author: wallisj
 * Created: July 17, 2008
 ********************************************************************
 * Local variables of program IPConfig
 ********************************************************************)
VAR
	ActBroadcastAddr : STRING[16];
	ActDefaultGateway : STRING[16];
	ActIPAddr : STRING[16];
	ActSubnetMask : STRING[16];
	CfgGetBroadcastAddr_0 : CfgGetBroadcastAddr;
	CfgGetDefaultGateway_0 : CfgGetDefaultGateway;
	CfgGetInaNode_0 : CfgGetInaNode;
	CfgGetIPAddr_0 : CfgGetIPAddr;
	CfgGetSubnetMask_0 : CfgGetSubnetMask;
	CfgSetBroadcastAddr_0 : CfgSetBroadcastAddr;
	CfgSetDefaultGateway_0 : CfgSetDefaultGateway;
	CfgSetIPAddr_0 : CfgSetIPAddr;
	CfgSetSubnetMask_0 : CfgSetSubnetMask;
	InaNodeNumber : USINT;
	ReadBroadcastAddr : BOOL;
	ReadBroadcastAddrError : UINT;
	ReadDefaultGateway : BOOL;
	ReadDefaultGatewayError : UINT;
	ReadEthernetSettings : BOOL;
	ReadInaNode : BOOL;
	ReadInaNodeError : UINT;
	ReadIPAddr : BOOL;
	ReadIPAddrError : UINT := 0;
	ReadSubnetMask : BOOL;
	ReadSubnetMaskError : UINT;
	ReBoot : BOOL;
	SetBroadcastAddr : STRING[16];
	SetDefaultGateway : STRING[16];
	SetIPAddr : STRING[16];
	SetSubnetMask : STRING[16];
	WriteBroadcastAddr : BOOL;
	WriteBroadcastAddrError : UINT;
	WriteDefaultGateway : BOOL;
	WriteDefaultGatewayError : UINT;
	WriteEthernetSettings : BOOL;
	WriteIPAddr : BOOL;
	WriteIPAddrError : UINT;
	WriteSubnetMask : BOOL;
	WriteSubnetMaskError : UINT;
END_VAR
```

### Program Logical/IPConfig/IPConfig (IEC) - Ethernet settings read/write

#### IPConfigInit.st - Initialization code
```iecst
(********************************************************************
 * COPYRIGHT --
 ********************************************************************
 * Program: IPConfig
 * File: IPConfigInit.st
 * Author: wallisj
 * Created: July 17, 2008
 ********************************************************************
 * Implementation of program IPConfig
 ********************************************************************)

PROGRAM _INIT

	ReadEthernetSettings := TRUE;

END_PROGRAM
```

#### IPConfigCyclic.st - Cyclic code
```iecst
(********************************************************************
 * COPYRIGHT --
 ********************************************************************
 * Program: IPConfig
 * File: IPConfigCyclic.st
 * Author: wallisj
 * Created: July 17, 2008
 ********************************************************************
 * Implementation of program IPConfig
 ********************************************************************)

PROGRAM _CYCLIC

(*----------------------------------------------------------------------------------*)
(* Flag control for reading the Ethernet settings									*)
(*----------------------------------------------------------------------------------*)
	IF (ReadEthernetSettings = TRUE) THEN
 		ReadInaNode 			:= TRUE;
		ReadIPAddr				:= TRUE;
		ReadSubnetMask			:= TRUE;
		ReadDefaultGateway		:= TRUE;
		ReadBroadcastAddr		:= TRUE;
		ReadEthernetSettings	:= FALSE;
	END_IF

(*----------------------------------------------------------------------------------*)
(* Flag control for writing the Ethernet settings									*)
(*----------------------------------------------------------------------------------*)
	IF (WriteEthernetSettings = TRUE) THEN
 		WriteIPAddr				:= TRUE;
		WriteSubnetMask			:= TRUE;
		WriteDefaultGateway		:= TRUE;
		WriteBroadcastAddr		:= TRUE;
		WriteEthernetSettings	:= FALSE;
	END_IF

(*----------------------------------------------------------------------------------*)
(* Read in the INA node number														*)
(*----------------------------------------------------------------------------------*)
	CfgGetInaNode_0.enable 		:= ReadInaNode;
	CfgGetInaNode_0.pDevice 	:= ADR('IF3');
 	CfgGetInaNode_0();

	IF(CfgGetInaNode_0.status = 0) THEN
		InaNodeNumber			:= CfgGetInaNode_0.InaNode;
		ReadInaNode				:= FALSE;
	ELSIF(CfgGetInaNode_0.status = 65534) THEN
		(* function block call disabled *)
	ELSIF(CfgGetInaNode_0.status = 65535) THEN
		(* function block busy *)
	ELSE
		(* error recording *)
		ReadInaNodeError 		:= CfgGetInaNode_0.status;
	END_IF

(*----------------------------------------------------------------------------------*)
(* Read in the IP address 															*)
(*----------------------------------------------------------------------------------*)
	CfgGetIPAddr_0.enable 		:= ReadIPAddr;
	CfgGetIPAddr_0.pDevice 		:= ADR('IF3');
	CfgGetIPAddr_0.pIPAddr		:= ADR(ActIPAddr);
 	CfgGetIPAddr_0.Len			:= 16;
 	CfgGetIPAddr_0();

	IF(CfgGetIPAddr_0.status = 0) THEN
		ReadIPAddr				:= FALSE;
	ELSIF(CfgGetIPAddr_0.status = 65534) THEN
		(* function block call disabled *)
	ELSIF(CfgGetIPAddr_0.status = 65535) THEN
		(* function block busy *)
	ELSE
		(* error recording *)
		ReadIPAddrError 		:= CfgGetIPAddr_0.status;
	END_IF

(*----------------------------------------------------------------------------------*)
(* Read in the subnet mask															*)
(*----------------------------------------------------------------------------------*)
	CfgGetSubnetMask_0.enable 		:= ReadSubnetMask;
	CfgGetSubnetMask_0.pDevice 		:= ADR('IF3');
	CfgGetSubnetMask_0.pSubnetMask	:= ADR(ActSubnetMask);
 	CfgGetSubnetMask_0.Len			:= 16;
 	CfgGetSubnetMask_0();

	IF(CfgGetSubnetMask_0.status = 0) THEN
		ReadSubnetMask				:= FALSE;
	ELSIF(CfgGetSubnetMask_0.status = 65534) THEN
		(* function block call disabled *)
	ELSIF(CfgGetSubnetMask_0.status = 65535) THEN
		(* function block busy *)
	ELSE
		(* error recording *)
		ReadSubnetMaskError 		:= CfgGetSubnetMask_0.status;
	END_IF

(*----------------------------------------------------------------------------------*)
(* Read in the gateway address														*)
(*----------------------------------------------------------------------------------*)
	CfgGetDefaultGateway_0.enable			:= ReadDefaultGateway;
	CfgGetDefaultGateway_0.pDevice 			:= ADR('IF3');
	CfgGetDefaultGateway_0.pGateway			:= ADR(ActDefaultGateway);
 	CfgGetDefaultGateway_0.Len				:= 16;
 	CfgGetDefaultGateway_0();

	IF(CfgGetDefaultGateway_0.status = 0) THEN
		ReadDefaultGateway					:= FALSE;
	ELSIF(CfgGetDefaultGateway_0.status = 65534) THEN
		(* function block call disabled *)
	ELSIF(CfgGetDefaultGateway_0.status = 65535) THEN
		(* function block busy *)
	ELSE
		(* error recording *)
		ReadDefaultGatewayError 			:= CfgGetDefaultGateway_0.status;
	END_IF

(*----------------------------------------------------------------------------------*)
(* Read in the broadcast address													*)
(*----------------------------------------------------------------------------------*)
	CfgGetBroadcastAddr_0.enable			:= ReadBroadcastAddr;
	CfgGetBroadcastAddr_0.pDevice 			:= ADR('IF3');
	CfgGetBroadcastAddr_0.pBroadcastAddr	:= ADR(ActBroadcastAddr);
 	CfgGetBroadcastAddr_0.Len				:= 16;
 	CfgGetBroadcastAddr_0();

	IF(CfgGetBroadcastAddr_0.status = 0) THEN
		ReadBroadcastAddr					:= FALSE;
	ELSIF(CfgGetBroadcastAddr_0.status = 65534) THEN
		(* function block call disabled *)
	ELSIF(CfgGetBroadcastAddr_0.status = 65535) THEN
		(* function block busy *)
	ELSE
		(* error recording *)
		ReadBroadcastAddrError 				:= CfgGetBroadcastAddr_0.status;
	END_IF

(*----------------------------------------------------------------------------------*)
(* Write the IP address 															*)
(*----------------------------------------------------------------------------------*)
	CfgSetIPAddr_0.enable 		:= WriteIPAddr;
	CfgSetIPAddr_0.pDevice 		:= ADR('IF3');
	CfgSetIPAddr_0.pIPAddr		:= ADR(SetIPAddr);
 	CfgSetIPAddr_0.Option		:= 1;
	(* Note set Option to 0 to make the value volatile and 1 to make it non volatile *)
 	CfgSetIPAddr_0();

	IF(CfgSetIPAddr_0.status = 0) THEN
		WriteIPAddr				:= FALSE;
	ELSIF(CfgSetIPAddr_0.status = 65534) THEN
		(* function block call disabled *)
	ELSIF(CfgSetIPAddr_0.status = 65535) THEN
		(* function block busy *)
	ELSE
		(* error recording *)
		WriteIPAddrError 		:= CfgSetIPAddr_0.status;
	END_IF

(*----------------------------------------------------------------------------------*)
(* Write the subnet mask															*)
(*----------------------------------------------------------------------------------*)
	CfgSetSubnetMask_0.enable 		:= WriteSubnetMask;
	CfgSetSubnetMask_0.pDevice 		:= ADR('IF3');
	CfgSetSubnetMask_0.pSubnetMask	:= ADR(SetSubnetMask);
 	CfgSetSubnetMask_0.Option		:= 1;
	(* Note set Option to 0 to make the value volatile and 1 to make it non volatile *)
 	CfgSetSubnetMask_0();

	IF(CfgSetSubnetMask_0.status = 0) THEN
		WriteSubnetMask				:= FALSE;
	ELSIF(CfgSetSubnetMask_0.status = 65534) THEN
		(* function block call disabled *)
	ELSIF(CfgSetSubnetMask_0.status = 65535) THEN
		(* function block busy *)
	ELSE
		(* error recording *)
		WriteSubnetMaskError 		:= CfgSetSubnetMask_0.status;
	END_IF

(*----------------------------------------------------------------------------------*)
(* Write the gateway address														*)
(*----------------------------------------------------------------------------------*)
	CfgSetDefaultGateway_0.enable			:= WriteDefaultGateway;
	CfgSetDefaultGateway_0.pDevice 			:= ADR('IF3');
	CfgSetDefaultGateway_0.pGateway			:= ADR(SetDefaultGateway);
 	CfgSetDefaultGateway_0.Option			:= 1;
 	(* Note set Option to 0 to make the value volatile and 1 to make it non volatile *)
	CfgSetDefaultGateway_0();

	IF(CfgSetDefaultGateway_0.status = 0) THEN
		WriteDefaultGateway					:= FALSE;
	ELSIF(CfgSetDefaultGateway_0.status = 65534) THEN
		(* function block call disabled *)
	ELSIF(CfgSetDefaultGateway_0.status = 65535) THEN
		(* function block busy *)
	ELSE
		(* error recording *)
		WriteDefaultGatewayError 			:= CfgSetDefaultGateway_0.status;
	END_IF

(*----------------------------------------------------------------------------------*)
(* Write the broadcast address														*)
(*----------------------------------------------------------------------------------*)
	CfgSetBroadcastAddr_0.enable			:= WriteBroadcastAddr;
	CfgSetBroadcastAddr_0.pDevice 			:= ADR('IF3');
	CfgSetBroadcastAddr_0.pBroadcastAddr	:= ADR(SetBroadcastAddr);
 	CfgSetBroadcastAddr_0.Option			:= 1;
 	(* Note set Option to 0 to make the value volatile and 1 to make it non volatile *)
	CfgSetBroadcastAddr_0();

	IF(CfgSetBroadcastAddr_0.status = 0) THEN
		WriteBroadcastAddr					:= FALSE;
	ELSIF(CfgSetBroadcastAddr_0.status = 65534) THEN
		(* function block call disabled *)
	ELSIF(CfgSetBroadcastAddr_0.status = 65535) THEN
		(* function block busy *)
	ELSE
		(* error recording *)
		WriteBroadcastAddrError				:= CfgSetBroadcastAddr_0.status;
	END_IF

(*----------------------------------------------------------------------------------*)
(* Reset the controller	- warm re-start												*)
(*----------------------------------------------------------------------------------*)
	IF (ReBoot = TRUE) THEN
 		SYSreset(1,1);
	END_IF

(*----------------------------------------------------------------------------------*)
(* End of task																		*)
(*----------------------------------------------------------------------------------*)
END_PROGRAM
```

### Package Logical/VisControl - Service visualisation control

### VisuControl.typ - Local data types
```iecst
(********************************************************************
 * COPYRIGHT --
 ********************************************************************
 * Program: VisuControl
 * File: VisuControl.typ
 * Author: nicke
 * Created: January 17, 2013
 ********************************************************************
 * Local data types of program VisuControl
 ********************************************************************)

TYPE
	CalcFreq_typ : 	STRUCT
		CurrentFreq : REAL; (*Current frequency*)
		NewFreq : REAL; (*New frequency*)
		NewSpeed : REAL; (*New speed*)
		CurrentSpeed : REAL; (*Current speed*)
		Disp : Status_enum := HIDE; (*Visu control*)
	END_STRUCT;
	CalcBelt_typ : 	STRUCT
		Unground : REAL; (*Unground size*)
		Current : REAL; (*Current preset*)
		New : REAL; (*New preset*)
		Adjust : REAL; (*Adjust delay by*)
		Disp : Status_enum := HIDE; (*Visu control*)
		Delay : BOOL; (*0 = OFF, 0 = ON*)
	END_STRUCT;
	INIT_typ : 	STRUCT
		TimeoutEnable : BOOL; (*Start initialisation delay*)
		TON : TON; (*Initialisation delay*)
		Progress : USINT; (*Progress bar value*)
	END_STRUCT;
	IP_typ : 	STRUCT
		Enable : Status_enum := HIDE; (*Enable IP Change*)
		ButtonEnable : Status_enum := HIDE; (*Enable button for IP Change*)
	END_STRUCT;
	Start_0_typ : 	STRUCT
		ResetEnable : Status_enum := HIDE; (*Show Inverter Reset Button*)
		Enable : Status_enum := HIDE; (*Show start information*)
		StatusSeam1 : Colour_enum := GREY; (*Seamer 1 Status Colour*)
		StatusSeam2 : Colour_enum := GREY; (*Seamer2 Status Colour*)
		StatusED : Colour_enum := GREY; (*Edge Deletion Status Colour*)
		TestEnable : Status_enum := HIDE; (*Show Test Buttons*)
	END_STRUCT;
	STATEREADY_enum :
		(
		WAIT := 0, (*Waiting for ready.*)
		READY_CONTROL := 1, (*Control circuit ready*)
		READY_SERVOS := 2, (*Servo systems ready*)
		READY_SEAMERS := 3, (*Grinding motors ready*)
		READY_CONTROL_SERVOS := 4, (*Control and Servos ready*)
		READY_CONTROL_SEAMERS := 5, (*Control and Grinding ready*)
		READY_ALL := 10 (*All systems ready.*)
		);
	Colour_enum :
		(
		BLACK := 0, (*Colour Black*)
		GREY := 7, (*Colour Grey*)
		WHITE := 15, (*Colour White*)
		RED := 45, (*Colour Red*)
		YELLOW := 46, (*Colour Yellow*)
		YELLOW_EVENT := 47, (*Event Yellow*)
		ORANGE_SDM := 49, (*SDM Orange*)
		RED_MENU := 87, (*Menu Red*)
		LILAC := 90, (*Lilac*)
		VIOLET_ACTIVE := 97, (*Selected Violet*)
		VIOLET := 98, (*Colour Violet*)
		GREEN_DARK := 180, (*Colour Dark Green*)
		GREEN := 184, (*Colour Green*)
		GREEN_OPTIONS := 185, (*Options Green*)
		GREEN1_ACTIVE := 191, (*Selected Green - Servo*)
		GREEN1 := 192, (*Colour Green - Servo*)
		LIGHTBLUE_ACTIVE := 196, (*Selected Light Blue*)
		LIGHTBLUE := 197, (*Colour Light Blue*)
		BLUE_ACTIVE := 4039, (*Selected Blue (199) with white (15) foreground*)
		BLUE := 4040, (*Colour Blue (200) with white(15) foreground*)
		GREY_ASHTON := 251, (*Ashton Grey*)
		ORANGE := 253, (*Colour Orange*)
		GREY_MIMIC := 255, (*Mimic Grey*)
		FONT_BLUE := 256,
		FONT_GREEN := 512,
		FONT_DARK_RED := 1024,
		FONT_MAGENTA := 1280,
		FONT_LIGHT_GREY := 1792,
		FONT_DARK_GREY := 2048,
		FONT_LIGHT_BLUE := 2816,
		FONT_WHITE := 3840,
		DROP_UNSELECTED := 3847, (*Foreground White (15) Background Grey (7)*)
		FONT_ORANGE := 10752,
		FONT_RED := 11520,
		FONT_YELLOW := 11776
		);
	Status_typ : 	STRUCT
		StatusSeamer : Colour_enum := RED; (*Seamer Status Colour*)
		StatusOffline : Colour_enum := RED; (*Offline Control Status Colour*)
		StatusServo : Colour_enum := RED; (*Imaging Status Colour*)
		StatusLaser : Colour_enum := RED; (*Robot Status Colour*)
		Enable : Status_enum := HIDE; (*Show status information*)
		TextYel : USINT := 0; (*Yellow Lamp text level*)
		TextGrn : USINT := 0; (*Green Lamp text level*)
		TextRed : USINT := 0; (*Red Lamp text level*)
		GrnLmp : Colour_enum := GREY; (*Green Lamp Colour*)
		YelLmp : Colour_enum := GREY; (*Yellow Lamp Colour (Shown as Blue)*)
		RedLmp : Colour_enum := GREY; (*Red Lamp Colour*)
		AlarmCount : USINT := 0; (*Alarm Count*)
		AlarmEnable : Status_enum := HIDE; (*Alarm display control*)
		WarningCount : USINT := 0; (*Warning Count*)
		WarningEnable : Status_enum := HIDE; (*Warning display control*)
	END_STRUCT;
	ESTOP_typ : 	STRUCT
		Confirm : ARRAY[0..4]OF BOOL; (*Visu control*)
		Disp : ARRAY[0..4]OF Status_enum; (*Visu control*)
		Recovery : BOOL; (*During recovery sequence*)
	END_STRUCT;
	Message_typ : 	STRUCT
		Text : STRING[75]; (*Message string to display. Controlled by NE*)
		Display : Status_enum := HIDE; (*Show or hide message.*)
	END_STRUCT;
	Visapi_typ : 	STRUCT
		READY : UINT := 0; (*VISAPI library control*)
		VC_HANDLE : UDINT := 0; (*VISAPI library control*)
		TOUCH : TouchAction := (0); (*VISAPI library control*)
		Status : UINT; (*VISAPI library control*)
	END_STRUCT;
	Vis_typ : 	STRUCT
		Page : PageControl_typ; (*Change sccreen control*)
		API : Visapi_typ; (*VISAPI library controls*)
		Init : INIT_typ; (*Screen Initialisation*)
		Message : Message_typ; (*NE Message display*)
		IP : IP_typ; (*IP screen control*)
		Start : Start_0_typ; (*Start screen control*)
		Status : Status_typ; (*Status screen control*)
		StepReady : STATEREADY_enum := WAIT; (*State Machine*)
		P10 : LayersNew_typ := (Index:=1,EnableIndex:=24); (*P10 Menu visualisation controls*)
		P11 : LayersNew_typ := (Index:=1,EnableIndex:=24); (*P11 Mimic visualisation controls*)
		P12 : LayersNew_typ := (Index:=1,EnableIndex:=24); (*P12 Options visualisation controls*)
		P13 : LayersNew_typ := (Index:=1,EnableIndex:=0); (*P13 Settings visualisation controls*)
		P13Drives : LayersNew_typ := (Index:=1,EnableIndex:=24); (*P13 Drives visualisation controls*)
		P13Delays : LayersNew_typ := (Index:=1,EnableIndex:=24); (*P13 Delays visualisation controls*)
		P13Servos : LayersNew_typ := (Index:=1,EnableIndex:=24); (*P13 Servos visualisation controls*)
		P13System : LayersNew_typ := (Index:=1,EnableIndex:=24); (*P13 System  visualisation controls*)
		P13Timeouts : LayersNew_typ := (Index:=1,EnableIndex:=24); (*P13 Timeouts visualisation controls*)
		P13Help1 : LayersNew_typ := (Index:=1,EnableIndex:=24); (*P13 Help visualisation controls 1*)
		P13Help2 : LayersNew_typ := (Index:=1,EnableIndex:=24); (*P13 Help visualisation controls 2*)
		P14Help : LayersNew_typ := (Index:=1,EnableIndex:=24); (*P14 Drives Help visualisation controls*)
		P14 : LayersNew_typ := (Index:=1,EnableIndex:=0); (*P14 Drives visualisation controls*)
		P14Layer : LayersNew_typ := (Index:=1,EnableIndex:=24); (*P14 Drives Layer visualisation controls*)
		P14Status : LayersNew_typ := (Index:=1,EnableIndex:=24); (*P14 Drives Status visualisation controls*)
		P15 : LayersNew_typ := (Index:=1,EnableIndex:=0); (*P15 Servos visualisation controls*)
		P15Layer : LayersNew_typ := (Index:=1,EnableIndex:=24); (*P15 Servos Layer visualisation controls*)
		P16 : LayersNew_typ := (Index:=1,EnableIndex:=0); (*P16 Remote visualisation controls*)
		P16Layer : LayersNew_typ := (Index:=1,EnableIndex:=24); (*P16 Remote Layer visualisation controls*)
		P20 : LayersNew_typ := (Index:=1,EnableIndex:=0); (*P20 Ashton Tech visualisation controls*)
		P30 : LayersNew_typ := (Index:=1,EnableIndex:=0); (*P30 Variables visualisation controls*)
		EMO : ESTOP_typ; (*Estop recovery controls*)
		HideAll : ARRAY[0..23]OF Status_enum := [24(HIDE)]; (*Hide all before case statements*)
		HeaderColour : Colour_enum; (*Header Bar Colour*)
		ConDisp : ARRAY[0..24]OF USINT; (*Conveyor text level control*)
		CalcBelt : CalcBelt_typ; (*Belt timings calculator*)
		CalcFreq : CalcFreq_typ; (*Frequency calculator*)
		FlipDisp1 : VisFlip_typ; (*Runtime control for warning Displays*)
		FlipDisp2 : VisFlip_typ; (*Runtime control for warning Displays*)
	END_STRUCT;
	VisBatch_typ : 	STRUCT
		Page : PageControl_typ; (*Change sccreen control*)
		API : Visapi_typ; (*VISAPI library controls*)
		P1 : LayersNew_typ := (Index:=1,EnableIndex:=24); (*P1 Batch Display visualisation controls*)
		P2 : LayersNew_typ := (Index:=1,EnableIndex:=24); (*P2 Batch List visualisation controls*)
		HideAll : ARRAY[0..23]OF Status_enum := [24(HIDE)]; (*Hide all before case statements*)
		Param : VisapiParam_typ;
		State : ScaleBatch_enum;
		Control : ScaleStateControl_typ;
		Displayed : Displayed_typ;
	END_STRUCT;
	ScaleStateControl_typ : 	STRUCT
		RowsIndex : USINT; (*Index for number of rows in batch*)
		RowIndex : USINT; (*Index for number of pieces in row*)
		RowWidthRaw : REAL; (*Extracted Row Width size - always extract from Loads.FurnaceExit.Rows[1].Row[0].Width - use to calculate y1 value for first piece in row*)
		WidthRaw : REAL; (*Extracted raw width of next piece*)
		LengthRaw : REAL; (*Extracted raw length of next piece*)
		WidthScaled : UINT; (*Scaled width of next piece*)
		LengthScaled : UINT; (*Scaled length of next piece*)
		WidthExtracted : BOOL; (*Set to TRUE when Width has been extracted from Loads.FurnaceExit.Rows[1].Row[0].Width*)
		X1Old : UINT; (*Last X1 value*)
		LongestOld : UINT; (*Scaled longest in previous row value*)
		LongestScaled : UINT; (*Scaled longest in row value*)
		GapLScaled : UINT; (*Scaled length gap*)
		GapWScaled : UINT; (*Scaled width gap*)
		RowWidthScaled : UINT; (*Scaled row width size*)
		Y1Old : UINT; (*Last Y1 value*)
		StrTemp : STRING[12]; (*Temporary register for text creation*)
		StrInt : INT; (*Temporary register for english text creation*)
		StrReal : REAL; (*Temporary register for english text creation*)
	END_STRUCT;
	Displayed_typ : 	STRUCT
		Index : UINT;
		Data : ARRAY[0..200]OF DisplayBatch_typ;
		RefreshIndex : UINT;
	END_STRUCT;
	ScaleBatch_enum :
		(
		RESET_WAIT := 0,
		CONFIRM_LOAD := 8,
		CONFIRM_CLEAR := 9,
		EXTRACT_VALUES := 10,
		CALCULATE_X1 := 11,
		CALCULATE_X2 := 12,
		CALCULATE_X3 := 13,
		CHECK_NEXT := 14,
		CALCULATE_Y1 := 15,
		CALCULATE_Y2 := 16,
		CALCULATE_Y3 := 17,
		REDRAW := 20,
		REFRESH := 21,
		REFRESH_RECTANGLE := 22,
		REFRESH_TEXTOUT1 := 23,
		REFRESH_TEXTOUT2 := 24,
		REFRESH_TEXTOUT3 := 25
		);
	ScaleBatch_typ : 	STRUCT
		RefX1 : ARRAY[0..1]OF lcrCurveByPoints_TabEntry_type;
		ScaleX1 : LCRCurveByPoints;
		RefY1 : ARRAY[0..1]OF lcrCurveByPoints_TabEntry_type;
		ScaleY1 : LCRCurveByPoints;
		RefWidth : ARRAY[0..1]OF lcrCurveByPoints_TabEntry_type;
		ScaleWidth : LCRCurveByPoints;
		RefLength : ARRAY[0..1]OF lcrCurveByPoints_TabEntry_type;
		ScaleLength : LCRCurveByPoints;
		RefGapW : ARRAY[0..1]OF lcrCurveByPoints_TabEntry_type;
		ScaleGapW : LCRCurveByPoints;
		RefGapL : ARRAY[0..1]OF lcrCurveByPoints_TabEntry_type;
		ScaleGapL : LCRCurveByPoints;
	END_STRUCT;
	DisplayBatch_typ : 	STRUCT
		x1 : UINT; (*Top left x co-ordinate*)
		y1 : UINT; (*Top left y co-ordinate*)
		width : UINT; (*Rect Width value*)
		height : UINT; (*Rect Height value*)
		str : STRING[19];
	END_STRUCT;
	VisapiParam_typ : 	STRUCT
		font1 : UINT; (*Textout font index*)
		font2 : UINT; (*Textout font index*)
		x1 : UINT; (*Top left x co-ordinate*)
		x2 : UINT; (*Top left x co-ordinate, Str[0]*)
		x3 : UINT; (*Top left x co-ordinate, Str[2]*)
		y1 : UINT; (*Top left y co-ordinate*)
		y2 : UINT; (*Top left y co-ordinate, Str[0]*)
		y3 : UINT; (*Top left y co-ordinate, Str[2]*)
		width : UINT; (*Rect Width value*)
		height : UINT; (*Rect Height value*)
		fill : USINT; (*Rect fill color index*)
		color : USINT; (*Rect border color index*)
		fore1 : USINT; (*Textout foreground color index*)
		fore2 : USINT; (*Textout foreground color index*)
		back : USINT; (*Textout background color index*)
		str : STRING[19]; (*Textout text to be output*)
	END_STRUCT;
	PageControl_typ : 	STRUCT
		Old : PAGE_enum; (*Visu control last scan page*)
		New : PAGE_enum; (*Visu control new page*)
		Current : PAGE_enum; (*Visu control current page*)
		Changed : BOOL; (*Page changed*)
	END_STRUCT;
	LayersNew_typ : 	STRUCT
		Layers : LayerRef_typ; (*Layer control*)
		Status1 : ARRAY[0..23]OF Status_enum := [24(HIDE)]; (*Enable controls array*)
		Status : ARRAY[0..23]OF Status_enum := [24(HIDE)]; (*Enable controls array*)
		Colour : ARRAY[0..23]OF Colour_enum; (*Colour control*)
		Old : USINT; (*Old index value*)
		New : USINT; (*New index value*)
		Changed : BOOL; (*Layer changed*)
		IndexMax : USINT;
		IndexMin : USINT;
		Index : USINT; (*Layer index*)
		EnableIndex : USINT; (*Enable Controls Index*)
	END_STRUCT;
	LayerRef_typ : 	STRUCT
		Button1 : VisuControl_enum;
		Button2 : VisuControl_enum;
		Button3 : VisuControl_enum;
		Button4 : VisuControl_enum;
		Button5 : VisuControl_enum;
		Button6 : VisuControl_enum;
		Button7 : VisuControl_enum;
		Button8 : VisuControl_enum;
		Button9 : VisuControl_enum;
		Help1 : Status_enum := HIDE;
		Help2 : Status_enum := HIDE;
		Help3 : Status_enum := HIDE;
		Help4 : Status_enum := HIDE;
		Help5 : Status_enum := HIDE;
		Help6 : Status_enum := HIDE;
		Help7 : Status_enum := HIDE;
		Help8 : Status_enum := HIDE;
		Help9 : Status_enum := HIDE;
		Layer1 : Status_enum := HIDE;
		Layer2 : Status_enum := HIDE;
		Layer3 : Status_enum := HIDE;
		Layer4 : Status_enum := HIDE;
		Layer5 : Status_enum := HIDE;
		Layer6 : Status_enum := HIDE;
		Layer7 : Status_enum := HIDE;
		Layer8 : Status_enum := HIDE;
		Layer9 : Status_enum := HIDE;
		Layer10 : Status_enum := HIDE;
		Layer11 : Status_enum := HIDE;
		Layer12 : Status_enum := HIDE;
		Layer13 : Status_enum := HIDE;
		Layer14 : Status_enum := HIDE;
		Layer15 : Status_enum := HIDE;
	END_STRUCT;
	PAGE_enum :
		(
		P00_INITIALIZE := 0,
		P10_MENU := 10,
		P11_MIMIC := 11,
		P12_OPTIONS := 12,
		P13_SETTINGS := 13,
		P14_DRIVES := 14,
		P15_SERVOS := 15,
		P16_RIO := 16,
		P17_ALARM := 17,
		P18_WARNING := 18,
		P19_EVENT := 19,
		P20_ASHTON_TECH := 20,
		P21_SDM := 21,
		P30_VARIABLES := 30,
		VIS_IDLE := 65535
		);
	VisuNew_typ : 	STRUCT
		Color : USINT; (*Appearance Color Datapoint*)
		PressedColor : USINT; (*Appearance Pressed Color Datapoint*)
		Index : USINT; (*Value Index Datapoint*)
		Min : USINT; (*Value Min Index Datapoint*)
		Max : USINT; (*Value Max Index Datapoint*)
		Value : USINT; (*Datapoint Value*)
		Status : Status_enum := HIDE; (*Runtime Status Datapoint*)
		P10 : LayersNew_typ := (Index:=1); (*P10 Menu visualisation controls*)
	END_STRUCT;
	Level_typ : 	STRUCT
		Delay : TON; (*Delay before confirm complete*)
		EnableSup : Status_enum := HIDE; (*Enable Supervisor level input*)
		EnableEng : Status_enum := HIDE; (*Enable Engineer level input*)
		EnableTech : Status_enum := HIDE; (*Enable Ashton Tech level input*)
		ResetEnable : Status_enum := HIDE; (*Enable Reset Defaults text*)
		EngEnable : Status_enum := HIDE; (*Enable Engineer change text*)
		SupEnable : Status_enum := HIDE; (*Enable Supervisor change text*)
		Enable : Status_enum := HIDE; (*Enable password input*)
		Entered : BOOL := FALSE; (*Password entered*)
		Eng : Status_enum := HIDE; (*Engineer level*)
		EngConfirm : BOOL := FALSE; (*Confirm new password entered*)
		EngNew : STRING[4]; (*New engineer password*)
		Level : Level_enum := OPERATOR; (*Level indicator*)
		Reset : BOOL := FALSE; (*Default reset*)
		Sup : Status_enum := HIDE; (*Supervisor level*)
		SupConfirm : BOOL := FALSE; (*Confirm new password entered*)
		SupNew : STRING[4]; (*New supervisor password*)
		EngRefused : Status_enum := HIDE; (*Display text  why engineering menu not available*)
		RefusedConfirm : BOOL; (*Confirm EngRefused*)
		ScreenTouch : BOOL; (*Turn on when screen touched.*)
		TechDelay : TON; (*Inactivity delay for password reset*)
		EngDelay : TON; (*Inactivity delay for password reset*)
		SupDelay : TON; (*Inactivity delay for password reset*)
		TechResetStart : BOOL; (*Start for reset delay*)
		EngResetStart : BOOL; (*Start for reset delay*)
		SupResetStart : BOOL; (*Start for reset delay*)
		BlockTech : BOOL; (*Block Tech reset delays when on specific screens*)
		BlockEng : BOOL; (*Block Engineering reset delays when on specific screens*)
		GTEngineerEnable : Status_enum := HIDE; (*Enable greater than Engineer level controls*)
		GTSupervisorEnable : Status_enum := HIDE; (*Enable greater than Supervisor level controls*)
		GTOperatorEnable : Status_enum := HIDE; (*Enable greater than Operator level controls*)
		TestModeEnable : Status_enum := HIDE; (*Test Mode enabled*)
		TestMode : Status_enum := HIDE; (*Test Mode enable*)
	END_STRUCT;
	CycleTest_typ : 	STRUCT
		Track001Time : UDINT := 500;
		Track002Time : UDINT := 500;
		Track003Time : UDINT := 3350;
		Track004Time : UDINT := 1200;
		Track09Time : UDINT := 3000;
		Track11Time : UDINT := 2230;
		Track12Time : UDINT := 340;
		Track413Time : UDINT := 1370;
		Track414Time : UDINT := 150;
		Track516Time : UDINT := 5010;
		Track517Time : UDINT := 1200;
		Track519Time : UDINT := 500;
		Track26Time : UDINT := 260;
		Track27Time : UDINT := 900;
		Track29Time : UDINT := 3000;
		Track31Time : UDINT := 1460;
		Track32Time : UDINT := 340;
		Track34Time : UDINT := 1310;
		Track35Time : UDINT := 1460;
		Track38Time : UDINT := 340;
		Track39Time : UDINT := 600;
		Track52Time : UDINT := 150;
		Track53Time : UDINT := 500;
		Track154Time : UDINT := 200;
		Track155Time : UDINT := 2600;
		Track256Time : UDINT := 1700;
		Track257Time : UDINT := 13000;
		Track558Time : UDINT := 7950;
		Track559Time : UDINT := 13000;
		Track64Time : UDINT := 10000;
		PivotTime : UDINT := 8000;
		TrackDelay : TON;
	END_STRUCT;
	Level_enum :
		(
		OPERATOR := 0,
		SUPERVISOR := 1,
		ENGINEER := 2,
		ASHTON_TECH := 3
		);
END_TYPE
```

### VisControl.var - Local variables
```iecst
(********************************************************************
 * COPYRIGHT --
 ********************************************************************
 * Program: Level
 * File: VisControll.var
 * Author: NickE
 * Created: January 18, 2013
 ********************************************************************
 * Local variables of program Level
 ********************************************************************)
VAR
	ScaleBatch : ScaleBatch_typ;
	VisBatch : VisBatch_typ;
	ServiceLevel : Level_typ;
	Level : Level_typ;
	ServiceVis : Vis_typ;
	Vis : Vis_typ;
END_VAR
```

### Package Logical/VisControl/HMIControl - Control for VisuNew

### Program Logical/VisControl/HMIControl/Level (IEC) - Password Level Control

#### Level.st - Cyclic code
```iecst
(********************************************************************
 * COPYRIGHT --
 ********************************************************************
 * Program: Level
 * File: Level.st
 * Author: NickE
 * Created: January 18, 2013
 ********************************************************************
 * Implementation of program Level
 ********************************************************************)

PROGRAM _INIT

	Vis.API.VC_HANDLE	:=	0	;

END_PROGRAM

PROGRAM _CYCLIC

	CASE Vis.Page.Current OF
		P00_INITIALIZE:
			//Init time - 3 sec
			Vis.Init.TimeoutEnable	:= TRUE					;
			Vis.Init.TON.IN			:= Vis.Init.TimeoutEnable	;
			Vis.Init.TON.PT			:= T#3000ms				;
			Vis.Init.TON ();

			Vis.Init.Progress	:=	UDINT_TO_USINT(TIME_TO_UDINT(Vis.Init.TON.ET) / 30);
			IF (Vis.Init.TON.Q) THEN
				//Switch to Menu Screen
				Vis.Page.New			:= 	P10_MENU	;
				Vis.Init.TimeoutEnable	:= 	FALSE		;
			END_IF
	END_CASE

	(*Hidden message control*)
	Vis.Message.Display	;
	Vis.Message.Text	;

	//GET TOUCH ACTION FROM SCREEN
	IF(Vis.API.READY <> 1) THEN
		Vis.API.VC_HANDLE := VA_Setup(1 , 'HMIXGA')	;

		IF(Vis.API.VC_HANDLE <> 0) THEN
			Vis.API.READY := 1	;
		END_IF
	END_IF

	IF(Vis.API.READY = 1) THEN
		IF(VA_Saccess(1,Vis.API.VC_HANDLE)= 0) THEN
			VA_GetTouchAction (1,Vis.API.VC_HANDLE,0,(ADR(Vis.API.TOUCH))) ;
			VA_Srelease(1,Vis.API.VC_HANDLE)	;
		END_IF
	END_IF

	IF(Vis.API.TOUCH.status = 1) THEN
		Level.ScreenTouch	:=	TRUE	;
	END_IF

	//PAGE CHANGE
	IF(Vis.Page.Current <> Vis.Page.Old) THEN
		Vis.Page.Changed	:=	TRUE	;
	ELSE
		Vis.Page.Changed	:=	FALSE	;
	END_IF
	Vis.Page.Old	:=	Vis.Page.Current;

	//HIDE DROP DOWN SCREENS
	IF(Vis.Page.Changed) THEN
		Vis.Start.Enable	:=	HIDE	;
		Vis.IP.Enable		:=	HIDE	;
		Vis.Status.Enable	:=	HIDE	;
		Level.Enable	:=	HIDE	;
		Level.EnableSup	:=	HIDE	;
		Level.EnableEng	:=	HIDE	;
//		Level.EnableTech	:=	HIDE	;
		IF NOT(Control.ESClear) THEN
			Vis.P11.EnableIndex		:=	24	;
		END_IF
		Vis.P12.EnableIndex		:=	24	;
	END_IF

	//HEADER BAR COLOUR DISPLAY
	CASE Vis.Page.Current OF
		P10_MENU:
			Vis.HeaderColour	:=	RED_MENU	;
		P11_MIMIC:
			Vis.HeaderColour	:=	GREY_MIMIC	;
		P12_OPTIONS:
			Vis.HeaderColour	:=	GREEN_OPTIONS	;
		P13_SETTINGS:
			Vis.HeaderColour	:=	BLUE	;
		P14_DRIVES:
			Vis.HeaderColour	:=	VIOLET	;
		P15_SERVOS:
			Vis.HeaderColour	:=	GREEN1	;
		P16_RIO:
			Vis.HeaderColour	:=	LIGHTBLUE	;
		P17_ALARM:
			Vis.HeaderColour	:=	RED	;
		P18_WARNING:
			Vis.HeaderColour	:=	ORANGE	;
		P19_EVENT:
			Vis.HeaderColour	:=	YELLOW_EVENT	;
		P20_ASHTON_TECH:
			Vis.HeaderColour	:=	GREY_ASHTON	;
		P21_SDM:
			Vis.HeaderColour	:=	ORANGE_SDM	;
		P30_VARIABLES:
			Vis.HeaderColour	:=	LILAC	;
	END_CASE

	//RESET SYSTEM PASSWORD
	IF NOT(SysPerm.PasswordDefault) THEN
		SysPerm.Password[0]		:= 	''		;
		SysPerm.Password[1]		:= 	'1'		;
		SysPerm.Password[2]		:= 	'5'		;
		SysPerm.Password[3]		:= 	'4046'	;
		SysPerm.PasswordDefault	:= 	TRUE	;
		Level.Delay.IN			:=	TRUE	;
		Level.Enable			:=	HIDE	;
		Level.ResetEnable		:=	SHOW	;
	END_IF

	//ENABLE SUPERVISOR LEVEL FOR TESTING
	Level.Level	:=	LIMIT(0,Level.Level,3)	;

	//Password control. Use level to enable different layers on screen rather than seperate screens.
	CASE Level.Level OF
		OPERATOR:
			Level.SupResetStart			:=	FALSE	;
			Level.EngResetStart			:=	FALSE	;
			Level.TechResetStart		:=	FALSE	;
			Level.EnableSup				:=	HIDE	;
			Level.EnableEng				:=	HIDE	;
			Level.EnableTech			:=	HIDE	;
			Level.GTOperatorEnable		:=	HIDE	;
			Level.GTSupervisorEnable	:=	HIDE	;
			Level.GTEngineerEnable		:=	HIDE	;
			Level.TestMode				:=	HIDE	;
			Control.Test				:=	FALSE	;
			Level.TestModeEnable		:=	HIDE	;
			MeterageReset1.Runtime := FB_HIDE;
			MeterageReset2.Runtime := FB_HIDE;
		SUPERVISOR:
			Level.SupResetStart			:=	TRUE	;
			Level.EnableSup				:=	Level.Enable	;
			Level.EnableEng				:=	HIDE	;
			Level.EnableTech			:=	HIDE	;
			Level.GTOperatorEnable		:=	SHOW	;
			Level.GTSupervisorEnable	:=	HIDE	;
			Level.GTEngineerEnable		:=	HIDE	;
			Level.TestMode				:=	HIDE	;
			Control.Test				:=	FALSE	;
			Level.TestModeEnable		:=	HIDE	;
			MeterageReset1.Runtime := FB_HIDE;
			MeterageReset2.Runtime := FB_HIDE;
			IF (Meterage1 = FB_SHOW) THEN
				MeterageReset1.Runtime := FB_SHOW;
			END_IF
			IF (Meterage2 = FB_SHOW) THEN
				MeterageReset2.Runtime := FB_SHOW;
			END_IF
		ENGINEER:
			Level.EngResetStart			:=	TRUE	;
			Level.EnableSup				:=	HIDE	;
			Level.EnableEng				:=	Level.Enable	;
			Level.EnableTech			:=	HIDE	;
			Level.GTOperatorEnable		:=	SHOW	;
			Level.GTSupervisorEnable	:=	SHOW	;
			Level.GTEngineerEnable		:=	HIDE	;
			Level.TestMode				:=	HIDE	;
			Level.TestModeEnable		:=	HIDE	;
			IF(Control.Empty) AND(Control.Achieved1) THEN
				Level.TestMode	:=	SHOW	;
			END_IF
			IF(Control.Test)THEN
				Level.TestModeEnable	:=	SHOW	;
				Level.TestMode	:=	SHOW	;
			END_IF
			MeterageReset1.Runtime := FB_SHOW;
			MeterageReset2.Runtime := FB_SHOW;
		ASHTON_TECH:
			Level.TechResetStart		:=	TRUE	;

			Level.EnableSup				:=	HIDE	;
			Level.EnableEng				:=	HIDE	;
			Level.EnableTech			:=	Level.Enable	;
			Level.GTOperatorEnable		:=	SHOW	;
			Level.GTSupervisorEnable	:=	SHOW	;
			Level.GTEngineerEnable		:=	SHOW	;
			Level.TestMode				:=	HIDE	;
			Level.TestModeEnable		:=	HIDE	;
			IF(Control.Empty) AND(Control.Achieved1) THEN
				Level.TestMode	:=	SHOW	;
			END_IF
			IF(Control.Test)THEN
				Level.TestModeEnable	:=	SHOW	;
				Level.TestMode	:=	SHOW	;
			END_IF
			MeterageReset1.Runtime := FB_SHOW;
			MeterageReset2.Runtime := FB_SHOW;
	END_CASE

	//Local Events List
	SysTemp.Events[95]	:=	Level.SupResetStart	;
	SysTemp.Events[96]	:=	Level.EngResetStart	;
	SysTemp.Events[97]	:=	Level.TechResetStart	;

	//RESET DROP DOWN SCREENS WHEN PASSWORD DISPLAYED
	IF EDGEPOS(Level.Enable = SHOW) THEN
		Vis.Start.Enable	:=	HIDE	;
		Vis.IP.Enable		:=	HIDE	;
		Vis.Status.Enable	:=	HIDE	;
	END_IF

	//ScreenTouch control for cancel password delay.
	Level.SupDelay.IN	:=	(Level.SupResetStart) AND NOT(Level.ScreenTouch)	;
	Level.SupDelay.PT	:=	t#2m	;
	Level.SupDelay();

	IF EDGEPOS(Level.SupDelay.Q) THEN
		Level.Level	:=	0	;
	END_IF

	Level.EngDelay.IN	:=	(Level.EngResetStart) AND NOT(Level.ScreenTouch) AND NOT(Level.BlockEng)	;
	Level.EngDelay.PT	:=	t#2m	;
	Level.EngDelay();

	IF EDGEPOS(Level.EngDelay.Q) THEN
		Level.Level	:=	0	;
	END_IF

	Level.TechDelay.IN	:=	(Level.TechResetStart) AND NOT(Level.ScreenTouch) AND NOT(Level.BlockTech)	;
	Level.TechDelay.PT	:=	t#2m	;
	Level.TechDelay();

	IF EDGEPOS(Level.TechDelay.Q) THEN
		Level.Level	:=	0	;
	END_IF

	Level.ScreenTouch	:=	FALSE	;

	IF(Control.Test) THEN
		Level.BlockEng	:=	TRUE	;
		Level.BlockTech	:=	TRUE	;
	ELSE
		Level.BlockEng	:=	FALSE	;
		Level.BlockTech	:=	FALSE	;
	END_IF

	IF(Vis.Page.Current >= P20_ASHTON_TECH) THEN
		Level.BlockTech	:=	TRUE	;
	ELSE
		Level.BlockTech	:=	FALSE	;
	END_IF

	IF(Control.Achieved1) AND(Control.Empty) THEN
		Level.EngRefused	:=	HIDE	;
	END_IF

	IF(Level.RefusedConfirm) THEN
		Level.EngRefused	:=	HIDE	;
		Level.Enable		:=	HIDE	;
	END_IF

	(*Change Password*)
	IF (Level.SupConfirm) THEN
		SysPerm.Password[1]	:= 	Level.SupNew	;
		Level.Delay.IN	:=	TRUE			;
		Level.SupEnable	:=	SHOW			;
	END_IF

	IF (Level.EngConfirm) THEN
		SysPerm.Password[2]	:= 	Level.EngNew	;
		Level.Delay.IN	:=	TRUE			;
		Level.EngEnable	:=	SHOW			;
	END_IF

	Level.Delay.PT	:=	T#2000ms	;
	Level.Delay ();

	IF(Level.Delay.Q) THEN
		Level.SupConfirm	:= 	FALSE	;
		Level.EngConfirm	:= 	FALSE	;
		Level.SupNew		:= 	''		;
		Level.EngNew		:= 	''		;
		Level.SupEnable		:=	HIDE	;
		Level.EngEnable		:=	HIDE	;
		Level.ResetEnable	:=	HIDE	;
		Level.Enable		:= 	HIDE	;
		Level.Delay.IN		:=	FALSE	;
	END_IF

	IF (Level.Entered) THEN
		Level.Enable	:= 	HIDE	;
		Level.Entered	:= 	FALSE	;
	END_IF

END_PROGRAM
```

### Program Logical/VisControl/HMIControl/Status (IEC) - Status bar screen control

#### Status.st - Cyclic code
```iecst
(********************************************************************
 * COPYRIGHT --
 ********************************************************************
 * Program: Status
 * File: Status.st
 * Author: NickE
 * Created: January 21, 2013
 ********************************************************************
 * Implementation of program Status
 ********************************************************************)

PROGRAM _CYCLIC

	//SEAMER CONTROL SYSTEM STATUS
	IF NOT(Control.Achieved1) THEN
		Vis.Status.StatusSeamer	:=	YELLOW		;
	END_IF

	IF(Control.Achieved1) THEN
		Vis.Status.StatusSeamer	:=	GREEN	;
	END_IF

	IF(Pause.Active) THEN
		Vis.Status.StatusSeamer	:=	Vis.Status.GrnLmp	;
	END_IF

	IF(Control.ESClear) THEN
		Vis.Status.StatusSeamer	:=	BLUE	;
	END_IF

	//OFFLINE CONTROL STATUS
	IF NOT(Control.Achieved2) THEN
		Vis.Status.StatusOffline	:=	YELLOW		;
	END_IF

	IF(Control.Achieved2) THEN
		Vis.Status.StatusOffline	:=	GREEN	;
	END_IF

	IF(Pause.Active) THEN
		Vis.Status.StatusOffline	:=	Vis.Status.GrnLmp	;
	END_IF

	//NUMBER OF ACTIVE WARNINGS
	Vis.Status.WarningCount		:=	0		;

	IF(Control.Warning) THEN
		Vis.Status.StatusSeamer	:=	ORANGE	;
		Vis.Status.WarningEnable	:=	SHOW	;
		FOR i:= 0 TO UINT_TO_INT(Warn.iMax) DO
			IF(Warn.Timeout[i]) THEN
				Vis.Status.WarningCount	:=	Vis.Status.WarningCount + 1	;
			END_IF
		END_FOR
	ELSE
		Vis.Status.WarningEnable	:=	HIDE	;
		Vis.Status.WarningCount		:=	0		;
	END_IF

	//NUMBER OF ACTIVE ALARMS
	Vis.Status.AlarmCount	:=	0		;

	IF(Control.Alarm) THEN
		Vis.Status.StatusSeamer	:=	RED		;
		Vis.Status.AlarmEnable	:=	SHOW	;
		FOR i := 0 TO 60 DO
			IF(SysTemp.Alarms[i]) THEN
				Vis.Status.AlarmCount	:=	Vis.Status.AlarmCount + 1	;
			END_IF
		END_FOR
	ELSE
		Vis.Status.AlarmEnable	:=	HIDE	;
		Vis.Status.AlarmCount	:=	0		;
	END_IF

	//SERVO STATUS
	IF NOT(Ax1.Error) AND NOT(Ax2.Error) AND NOT(Ax3.Error) THEN
		Vis.Status.StatusServo	:=	GREEN	;
	ELSE
		Vis.Status.StatusServo	:=	YELLOW	;
	END_IF
	IF(Ax1.Error) OR(Ax2.Error) OR(Ax3.Error) THEN
		Vis.Status.StatusServo	:=	RED	;
	END_IF

	//LASER STATUS
	IF(S56Lever.In) THEN
		Vis.Status.StatusLaser	:=	GREEN	;
	ELSE
		Vis.Status.StatusLaser	:=	YELLOW	;
	END_IF

	//LIGHTSTACK COLOURS
	IF(Control.RedLmp) THEN
		Vis.Status.RedLmp	:=	RED		;
		Vis.Status.TextRed	:=	1		;
	ELSE
		Vis.Status.RedLmp	:=	GREY	;
		Vis.Status.TextRed	:=	0		;
	END_IF

	IF(Control.GrnLmp) THEN
		Vis.Status.GrnLmp	:=	GREEN	;
		Vis.Status.TextGrn	:=	1		;
		IF(Pause.Active) THEN
			Vis.Status.TextGrn	:=	2	;
		END_IF
	ELSE
		Vis.Status.GrnLmp	:=	GREY	;
		Vis.Status.TextGrn	:=	0		;
		IF(Pause.Active) THEN
			Vis.Status.TextGrn	:=	2	;
		END_IF
	END_IF

	IF(Control.YelLmp) THEN
		Vis.Status.YelLmp	:=	BLUE	;
		Vis.Status.TextYel	:=	1		;
	ELSE
		Vis.Status.YelLmp	:=	GREY	;
		Vis.Status.TextYel	:=	0		;
	END_IF

	//RESET DROP DOWN SCREENS WHEN STATUS DISPLAYED
	IF EDGEPOS(Vis.Status.Enable = SHOW) THEN
		Vis.Start.Enable	:=	HIDE	;
		Vis.IP.Enable		:=	HIDE	;
		Level.Enable	:=	HIDE	;
		Level.EnableSup	:=	HIDE	;
		Level.EnableEng	:=	HIDE	;
		Level.EnableTech	:=	HIDE	;
	END_IF

END_PROGRAM
```

### Program Logical/VisControl/HMIControl/Start (IEC) - Start visualisation control

#### Start.st - Cyclic code
```iecst
(********************************************************************
 * COPYRIGHT --
 ********************************************************************
 * Program: Start
 * File: Start.st
 * Author: nicke
 * Created: January 21, 2013
 ********************************************************************
 * Implementation of program Start
 ********************************************************************)

PROGRAM _CYCLIC

	Vis.Start.ResetEnable	:= HIDE	;

	//STATUS LIGHTS FOR SEAMER 1
	IF(SeamersII.AutoStart[1]) THEN
		Vis.Start.StatusSeam1	:=	GREEN	;
	ELSE
		Vis.Start.StatusSeam1	:=	GREEN_DARK	;
	END_IF

	IF(SeamersII.Enable[1]) AND NOT(SeamersII.AutoStart[1]) THEN
		Vis.Start.StatusSeam1	:=	YELLOW	;
	END_IF

	IF(MS1Belt1.Trip) THEN
		Vis.Start.StatusSeam1	:=	RED	;
	ELSIF(MS2Belt2.Trip) THEN
		Vis.Start.StatusSeam1	:=	RED	;
	ELSIF(MS3Belt3.Trip) THEN
		Vis.Start.StatusSeam1	:=	RED	;
	ELSIF(MS4Belt4.Trip) THEN
		Vis.Start.StatusSeam1	:=	RED	;
	ELSIF(MS9Vac1.Trip) THEN
		Vis.Start.StatusSeam1	:=	RED	;
	ELSIF(MS11Vac3.Trip) THEN
		Vis.Start.StatusSeam1	:=	RED	;
	ELSIF(MS23Vac5.Trip) THEN
		Vis.Start.StatusSeam1	:=	RED	;
	ELSIF(MS24Vac6.Trip) THEN
		Vis.Start.StatusSeam1	:=	RED	;
	END_IF

	//STATUS LIGHTS FOR SEAMER 2
	IF(SeamersII.AutoStart[2]) THEN
		Vis.Start.StatusSeam2	:=	GREEN	;
	ELSE
		Vis.Start.StatusSeam2	:=	GREEN_DARK	;
	END_IF

	IF(SeamersII.Enable[2]) AND NOT(SeamersII.AutoStart[2]) THEN
		Vis.Start.StatusSeam2	:=	YELLOW	;
	END_IF

	IF(MS5Belt5.Trip) THEN
		Vis.Start.StatusSeam2	:=	RED	;
	ELSIF(MS6Belt6.Trip) THEN
		Vis.Start.StatusSeam2	:=	RED	;
	ELSIF(MS7Belt7.Trip) THEN
		Vis.Start.StatusSeam2	:=	RED	;
	ELSIF(MS8Belt8.Trip) THEN
		Vis.Start.StatusSeam2	:=	RED	;
	ELSIF(MS10Vac2.Trip) THEN
		Vis.Start.StatusSeam2	:=	RED	;
	ELSIF(MS12Vac4.Trip) THEN
		Vis.Start.StatusSeam2	:=	RED	;
	ELSIF(MS25Vac7.Trip) THEN
		Vis.Start.StatusSeam2	:=	RED	;
	ELSIF(MS26Vac8.Trip) THEN
		Vis.Start.StatusSeam2	:=	RED	;
	END_IF

	Control.Auto := NOT(Control.Test) ;

	IF EDGEPOS(Control.EStop1) AND(Control.Test) THEN
		Control.Test	:=	FALSE	;
		Vis.Start.Enable	:=	HIDE	;
	END_IF

END_PROGRAM
```

### Program Logical/VisControl/HMIControl/Page10 (IEC) - Menu screen

#### Page10.st - Cyclic code
```iecst
(********************************************************************
 * COPYRIGHT --
 ********************************************************************
 * Program: Page10
 * File: Page10.st
 * Author: NickE
 * Created: January 31, 2013
 ********************************************************************
 * Implementation of program Page10
 ********************************************************************)

PROGRAM _CYCLIC

	//MENU SCREEN
	Vis.P10.Status[0]	:=	HIDE	;
	Vis.P10.Status[1]	:=	HIDE	;
	Vis.P10.Status[2]	:=	HIDE	;
	Vis.P10.Status[3]	:=	HIDE	;
	Vis.P10.Status[4]	:=	HIDE	;
	Vis.P10.Status[5]	:=	HIDE	;
	Vis.P10.Status[6]	:=	HIDE	;
	Vis.P10.Status[7]	:=	HIDE	;
	Vis.P10.Status[8]	:=	HIDE	;
	Vis.P10.Status[9]	:=	HIDE	;
	Vis.P10.Status[10]	:=	HIDE	;

	CASE Vis.P10.EnableIndex OF
		0:
			Vis.P10.Status[0]	:=	SHOW	;
		1:
			Vis.P10.Status[1]	:=	SHOW	;
		2:
			Vis.P10.Status[2]	:=	SHOW	;
		3:
			Vis.P10.Status[3]	:=	SHOW	;
		4:
			Vis.P10.Status[4]	:=	SHOW	;
		5:
			Vis.P10.Status[5]	:=	SHOW	;
		6:
			Vis.P10.Status[6]	:=	SHOW	;
		7:
			Vis.P10.Status[7]	:=	SHOW	;
		8:
			Vis.P10.Status[8]	:=	SHOW	;
		9:
			Vis.P10.Status[9]	:=	SHOW	;

	END_CASE

END_PROGRAM
```

### Program Logical/VisControl/HMIControl/Page11 (IEC) - Mimic screen

#### Page11.st - Cyclic code
```iecst
(********************************************************************
 * COPYRIGHT --
 ********************************************************************
 * Program: Page11
 * File: Page11.st
 * Author: NickE
 * Created: January 31, 2013
 ********************************************************************
 * Implementation of program Page11
 ********************************************************************)

PROGRAM _CYCLIC

    //MIMIC SCREEN
    memcpy(ADR(Vis.P11.Status),ADR(Vis.HideAll),SIZEOF(Vis.HideAll));
    memcpy(ADR(Vis.P11.Status1),ADR(Vis.HideAll),SIZEOF(Vis.HideAll));
    //DISPLAY TRACK BLOCK CONDITION CONTROL
    Vis.P11.Layers.Layer1 := HIDE ;
    Vis.P11.Layers.Layer2 := HIDE ;
    Vis.P11.Layers.Layer3 := HIDE ;
    Vis.P11.Layers.Layer4 := HIDE ;
    Vis.P11.Layers.Layer5 := HIDE ;
    Vis.P11.Layers.Layer6 := HIDE ;
    Vis.P11.Layers.Layer7 := HIDE ;
    Vis.P11.Layers.Layer8 := HIDE ;
    Vis.P11.Layers.Layer9 := HIDE ;
    Vis.P11.Layers.Layer10 := HIDE ;
    Vis.P11.Layers.Layer11 := HIDE ;
    Vis.P11.Layers.Layer12 := HIDE ;
    Vis.P11.Layers.Layer13 := HIDE ;
    Vis.P11.Layers.Layer14 := HIDE ;
    Vis.P11.Layers.Layer15 := HIDE ;

    CASE Vis.P11.EnableIndex OF
        0:
            Vis.P11.Status[0] := SHOW ;
            IF(Level.Level > OPERATOR) AND(Tracking20.Busy) THEN
                Vis.P11.Status1[0] := SHOW ;
            END_IF
            IF(Track208.Active) AND(Tracking20.Blocked) THEN
                Vis.P11.Layers.Layer1 := SHOW ;
            END_IF
        1:
            Vis.P11.Status[1] := SHOW ;
            IF(Level.Level > OPERATOR) AND(Tracking30.Busy) THEN
                Vis.P11.Status1[1] := SHOW ;
            END_IF
			IF(Track302.Active) AND(Tracking30.Blocked) THEN
				Vis.P11.Layers.Layer2 := SHOW ;
			END_IF
        2:
            Vis.P11.Status[2] := SHOW ;
            IF(Level.Level > OPERATOR) AND(Tracking40.Busy) THEN
                Vis.P11.Status1[2] := SHOW ;
            END_IF
			IF(Track402.Active) AND(Tracking40.Blocked) THEN
				Vis.P11.Layers.Layer3 := SHOW ;
			END_IF
			IF(Level.Level > OPERATOR) AND(Tracking41.Busy) THEN
				Vis.P11.Status1[3] := SHOW ;
			END_IF
        3:
            Vis.P11.Status[3] := SHOW ;
            IF(Level.Level > OPERATOR) AND(Tracking50.Busy) THEN
                Vis.P11.Status1[4] := SHOW ;
            END_IF
			IF(Level.Level > OPERATOR) AND(Tracking80.Busy) THEN
				Vis.P11.Status1[5] := SHOW ;
			END_IF
			IF(Level.Level > OPERATOR) AND(Tracking51.Busy) THEN
				Vis.P11.Status[13] := SHOW ;
			END_IF
			IF(Track513.Active) AND(Tracking51.Blocked) THEN
				Vis.P11.Layers.Layer11 := SHOW ;
			END_IF
		4:
			Vis.P11.Status[4] := SHOW ;
			IF(Level.Level > OPERATOR) AND(Tracking60.Busy) THEN
				Vis.P11.Status1[6] := SHOW ;
			END_IF
			IF(Track603.Active) AND(Tracking60.Blocked) THEN
				Vis.P11.Layers.Layer4 := SHOW ;
			END_IF
			IF(Level.Level > OPERATOR) AND(Tracking70.Busy) THEN
				Vis.P11.Status1[7] := SHOW ;
			END_IF
			IF(Level.Level > OPERATOR) AND(Tracking81.Busy) THEN
				Vis.P11.Status1[8] := SHOW ;
			END_IF
			IF(Track812.Active) AND(Tracking81.Blocked) THEN
				Vis.P11.Layers.Layer5 := SHOW ;
			END_IF
			IF(Level.Level > OPERATOR) AND(Tracking82.Busy) THEN
				Vis.P11.Status1[9] := SHOW ;
			END_IF
			IF(Track521.Active) AND(Tracking52.Blocked) THEN
				Vis.P11.Layers.Layer12 := SHOW ;
			END_IF
			IF(Level.Level > OPERATOR) AND(Tracking52.Busy) THEN
				Vis.P11.Status1[13] := SHOW ;
			END_IF
		5:
			Vis.P11.Status[5] := SHOW ;
			IF(Level.Level > OPERATOR) AND(Tracking00.Busy) THEN
				Vis.P11.Status1[10] := SHOW ;
			END_IF
			IF(Track005.Active) AND(Tracking00.Blocked) THEN
				Vis.P11.Layers.Layer6 := SHOW ;
			END_IF
			IF(Track004.Active) AND(Ax1.Block) THEN
				Vis.P11.Layers.Layer7 := SHOW ;
			END_IF
		6:
			Vis.P11.Status[6] := SHOW ;
			IF(Level.Level > OPERATOR) AND(Tracking10.Busy) THEN
				Vis.P11.Status1[11] := SHOW ;
			END_IF
			IF(Track108.Active) AND(Tracking10.Blocked) THEN
				Vis.P11.Layers.Layer8 := SHOW ;
			END_IF
		7:
			Vis.P11.Status[7] := SHOW ;
			IF(Level.Level > OPERATOR) AND(Tracking11.Busy) THEN
				Vis.P11.Status1[12] := SHOW ;
			END_IF
			IF(Track115.Active) AND(Tracking11.Blocked) THEN
				Vis.P11.Layers.Layer9 := SHOW ;
			END_IF
			IF(Track114.Active) AND(Ax2.Block) THEN
				Vis.P11.Layers.Layer10 := SHOW ;
			END_IF
		8:
			Vis.P11.Status[8] := SHOW ;
			IF(Reset.Count) THEN
				Reset.Grind := TRUE ;
                Reset.Time := TRUE ;
            ELSE
                Reset.Grind := FALSE ;
                Reset.Time := FALSE ;
            END_IF
		9:
			Vis.P11.Status[9]	:=	SHOW	;
			IF((Track501.Active) OR(Track601.Active)) AND NOT((Tracking00.Busy) OR(Tracking10.Busy) OR(Tracking11.Busy) OR(Tracking20.Busy) OR(Tracking40.Busy) OR(Tracking30.Busy) OR(Tracking41.Busy) OR(Tracking70.Busy)) THEN //CHANGE TRACKING REGISTER AS REQUIRED
				Vis.P11.Status1[17]	:=	SHOW	;
			END_IF
		10:
			Vis.P11.Status[10]	:=	SHOW	;
		20:
			Vis.P11.Status[20]	:=	SHOW	;
			Vis.Start.Enable	:=	HIDE	;
		21:
			Vis.P11.Status[21]	:=	SHOW	;
		22:
			Vis.P11.Status[22]	:=	SHOW	;
	END_CASE

	IF NOT(Control.Achieved1) THEN
		Vis.P11.Status[16] :=	SHOW	;
	END_IF
	IF NOT(Control.Achieved2) THEN
		Vis.P11.Status[17] :=	SHOW	;
	END_IF
	IF NOT(WashRun.In) THEN
		Vis.P11.Status[18] :=	SHOW	;
	END_IF
	IF NOT(FurnReady.Int) THEN
		Vis.P11.Status[19] :=	SHOW	;
	END_IF
	IF NOT(AGVReady.In)THEN
		Vis.P11.Status[23] :=	SHOW	;
	END_IF
	IF(S57Lever.Int) THEN
		Vis.P11.Status[15] := SHOW ;
	END_IF
	IF(S58Lever.Int) THEN
		Vis.P11.Status[14] := SHOW ;
	END_IF

	//INFORMATION DISPLAY CONTROL
	IF Grind1.TotalMUpp > 0 THEN
		GrindDisp1.TotalDisp	:= 	SHOW	;
	ELSE
		GrindDisp1.TotalDisp	:= 	HIDE	;
	END_IF

	IF Grind2.TotalMUpp > 0 THEN
		GrindDisp2.TotalDisp	:= 	SHOW	;
	ELSE
		GrindDisp2.TotalDisp	:= 	HIDE	;
	END_IF

	IF Grind1.ShiftMUpp > 0 THEN
		GrindDisp1.ShiftDisp	:= 	SHOW	;
	ELSE
		GrindDisp1.ShiftDisp	:= 	HIDE	;
	END_IF

	IF Grind2.ShiftMUpp > 0 THEN
		GrindDisp2.ShiftDisp	:= 	SHOW	;
	ELSE
		GrindDisp2.ShiftDisp	:= 	HIDE	;
	END_IF

	//SENSOR BLOCK DISP
	S1Photo.BlockDisp := HIDE ;
	S2Photo.BlockDisp := HIDE ;
	S3Photo.BlockDisp := HIDE ;
	S4Photo.BlockDisp := HIDE ;
	S5Photo.BlockDisp := HIDE ;
	S6Photo.BlockDisp := HIDE ;
	S7Photo.BlockDisp := HIDE ;
	S8Photo.BlockDisp := HIDE ;
	S9Photo.BlockDisp := HIDE ;
	S12Photo.BlockDisp := HIDE ;
	S13Photo.BlockDisp := HIDE ;
	S14Photo.BlockDisp := HIDE ;
	S15Photo.BlockDisp := HIDE ;
	S16Photo.BlockDisp := HIDE ;
	S17Photo.BlockDisp := HIDE ;
	S18Photo.BlockDisp := HIDE ;
	S19Photo.BlockDisp := HIDE ;
	S20Photo.BlockDisp := HIDE ;
	S21Photo.BlockDisp := HIDE ;
	S50Reed.BlockDisp := HIDE ;
	IF(Tracking00.Blocks[9]) AND(Track005.Active) AND NOT(Tracking00.BlockInhib) THEN
		S3Photo.BlockDisp := SHOW ;
		Tracking00.Blocks[9] := FALSE ;
	END_IF
	IF(Tracking00.Blocks[10]) AND(Track005.Active) AND NOT(Tracking00.BlockInhib) THEN
		S4Photo.BlockDisp := SHOW ;
		Tracking00.Blocks[10] := FALSE ;
	END_IF
	IF(Tracking00.Blocks[12]) AND(Track005.Active) AND NOT(Tracking00.BlockInhib) THEN
		S50Reed.BlockDisp := SHOW ;
		Tracking00.Blocks[12] := FALSE ;
	END_IF
	IF(Tracking10.Blocks[9]) AND(Track108.Active) AND NOT(Tracking11.Busy) THEN
		S5Photo.BlockDisp := SHOW ;
		Tracking10.Blocks[9] := FALSE ;
	END_IF
	IF(Tracking10.Blocks[10]) AND(Track108.Active) AND NOT(Tracking11.Busy) THEN
		S6Photo.BlockDisp := SHOW ;
		Tracking10.Blocks[10] := FALSE ;
	END_IF
	IF(Tracking10.Blocks[11]) AND(Track108.Active) AND NOT(Tracking11.Busy) THEN
		S7Photo.BlockDisp := SHOW ;
		Tracking10.Blocks[11] := FALSE ;
	END_IF
	IF(Tracking11.Blocks[9]) AND(Track115.Active) AND NOT(Tracking11.BlockInhib) THEN
		S8Photo.BlockDisp := SHOW ;
		Tracking11.Blocks[9] := FALSE ;
	END_IF
	IF(Tracking11.Blocks[10]) AND(Track115.Active) AND NOT(Tracking11.BlockInhib) THEN
		S12Photo.BlockDisp := SHOW ;
		Tracking11.Blocks[10] := FALSE ;
	END_IF
	IF(Tracking20.Blocks[9]) AND(Track208.Active) AND NOT(Track302.Active) THEN
		S14Photo.BlockDisp := SHOW ;
		Tracking20.Blocks[9] := FALSE ;
	END_IF
	IF(Tracking20.Blocks[10]) AND(Track208.Active) AND NOT(Track302.Active) THEN
		S15Photo.BlockDisp := SHOW ;
		Tracking20.Blocks[10] := FALSE ;
	END_IF
	IF(Tracking30.Blocks[9]) AND(Track302.Active) AND NOT(Track402.Active) THEN
		S16Photo.BlockDisp := SHOW ;
		Tracking30.Blocks[9] := FALSE ;
	END_IF
	IF(Tracking30.Blocks[10]) AND(Track302.Active) THEN
		S17Photo.BlockDisp := SHOW ;
		Tracking30.Blocks[10] := FALSE ;
	END_IF
	IF(Tracking40.Blocks[9]) AND(Track402.Active) THEN
		S17Photo.BlockDisp := SHOW ;
		Tracking40.Blocks[9] := FALSE ;
	END_IF
	IF(Tracking40.Blocks[10]) AND(Track402.Active) THEN
		S18Photo.BlockDisp := SHOW ;
		Tracking40.Blocks[10] := FALSE ;
	END_IF
	IF(Tracking50.Blocks[9]) AND(Track503.Active) THEN
		S19Photo.BlockDisp := SHOW ;
		Tracking50.Blocks[9] := FALSE ;
	END_IF
	IF(Tracking50.Blocks[10]) AND(Track503.Active) THEN
		S20Photo.BlockDisp := SHOW ;
		Tracking50.Blocks[10] := FALSE ;
	END_IF
	IF(Tracking50.Blocks[11]) AND(Track503.Active) AND NOT(Track603.Active) THEN
		S21Photo.BlockDisp := SHOW ;
		Tracking50.Blocks[11] := FALSE ;
	END_IF
	IF(Tracking80.Blocks[9]) AND(Track803.Active) THEN
		S19Photo.BlockDisp := SHOW ;
		Tracking80.Blocks[9] := FALSE ;
	END_IF

END_PROGRAM
```

### Program Logical/VisControl/HMIControl/Page12 (IEC) - Options screen

#### Page12.st - Cyclic code
```iecst
(********************************************************************
 * COPYRIGHT --
 ********************************************************************
 * Program: Page12
 * File: Page12.st
 * Author: NickE
 * Created: January 31, 2013
 ********************************************************************
 * Implementation of program Page12
 ********************************************************************)

PROGRAM _CYCLIC

	//OPTIONS SCREEN
	Vis.P12.Status[0]	:=	HIDE	;
	Vis.P12.Status[1]	:=	HIDE	;
	Vis.P12.Status[2]	:=	HIDE	;
	Vis.P12.Status[3]	:=	HIDE	;
	Vis.P12.Status[4]	:=	HIDE	;
	Vis.P12.Status[5]	:=	HIDE	;
	Vis.P12.Status[6]	:=	HIDE	;
	Vis.P12.Status[7]	:=	HIDE	;
	Vis.P12.Status[8]	:=	HIDE	;
	Vis.P12.Status[9]	:=	HIDE	;
	Vis.P12.Status[10]	:=	HIDE	;
	Vis.P12.Status[11]	:=	HIDE	;

	CASE Vis.P12.EnableIndex OF
		0:
			Vis.P12.Status[0]	:=	SHOW	;
		1:
			Vis.P12.Status[1]	:=	SHOW	;
		2:
			Vis.P12.Status[2]	:=	SHOW	;
		3:
			Vis.P12.Status[3]	:=	SHOW	;
		4:
			Vis.P12.Status[4]	:=	SHOW	;
		5:
			Vis.P12.Status[5]	:=	SHOW	;
		6:
			Vis.P12.Status[6]	:=	SHOW	;
		7:
			Vis.P12.Status[7]	:=	SHOW	;
		8:
			Vis.P12.Status[8]	:=	SHOW	;
		9:
			Vis.P12.Status[9]	:=	SHOW	;
		10:
			Vis.P12.Status[10]	:=	SHOW	;
	END_CASE
	IF(Level.Level > OPERATOR)THEN
		Vis.P12.Status[9]	:=	SHOW	;
	END_IF

	IF (Control.Achieved1) THEN
		Sol20DT1.Auto	:=	FALSE	;
		Sol21DT2.Auto	:=	FALSE	;
		Sol22DT3.Auto	:=	FALSE	;
		Sol23DT4.Auto	:=	FALSE	;
	END_IF

	IF(Sol20DT1.Auto) THEN
		Sol21DT2.Auto	:=	TRUE	;
		Sol22DT3.Auto	:=	TRUE	;
		Sol23DT4.Auto	:=	TRUE	;
	ELSE
		Sol21DT2.Auto	:=	FALSE	;
		Sol22DT3.Auto	:=	FALSE	;
		Sol23DT4.Auto	:=	FALSE	;
	END_IF

	//DISABLE CHANGING BATCHING MODES UNTIL LINE IS EMPTY
	IF(Control.Empty) THEN
		Vis.P12.Status[11]	:=	SHOW	;
	END_IF

	//HIGHLIGHT SELECTED FURNACE CLEAR SIGNAL MODE COLOUR
	CASE LoadPerm.FurnClear OF
		0:
			Vis.P12.Colour[5]	:=	WHITE			;
			Vis.P12.Colour[6]	:=	DROP_UNSELECTED	;
		1:
			Vis.P12.Colour[5]	:=	DROP_UNSELECTED	;
			Vis.P12.Colour[6]	:=	WHITE			;
	END_CASE

END_PROGRAM
```

### Program Logical/VisControl/HMIControl/Page13 (IEC) - Settings screen
